LIN {X 0,Y 375.934,Z 136.466,A -85,B 0,C 180,E1 -12378.399,E2 -12378.399} C_VEL
LIN {X 0,Y 375.973,Z 136.465,A -85,B 0,C 180,E1 -12381.73,E2 -12381.73} C_VEL
LIN {X 0,Y 375.981,Z 136.466,A -85,B 0,C 180,E1 -12385.333,E2 -12385.333} C_VEL
LIN {X 0,Y 375.958,Z 136.463,A -85,B 0,C 180,E1 -12388.438,E2 -12388.438} C_VEL
LIN {X 0,Y 375.997,Z 136.458,A -85,B 0,C 180,E1 -12392.142,E2 -12392.142} C_VEL
LIN {X 0,Y 376.007,Z 136.459,A -85,B 0,C 180,E1 -12394.539,E2 -12394.539} C_VEL
LIN {X 0,Y 375.964,Z 136.462,A -85,B 0,C 180,E1 -12398.046,E2 -12398.046} C_VEL
LIN {X 0,Y 376.01,Z 136.457,A -85,B 0,C 180,E1 -12401.473,E2 -12401.473} C_VEL
LIN {X 0,Y 376.06,Z 136.455,A -85,B 0,C 180,E1 -12404.833,E2 -12404.833} C_VEL
LIN {X 0,Y 376.052,Z 136.454,A -85,B 0,C 180,E1 -12408.137,E2 -12408.137} C_VEL
LIN {X 0,Y 376.22,Z 136.432,A -85,B 0,C 180,E1 -12411.919,E2 -12411.919} C_VEL
LIN {X 0,Y 376.17,Z 136.439,A -85,B 0,C 180,E1 -12414.64,E2 -12414.64} C_VEL
LIN {X 0,Y 376.353,Z 136.417,A -85,B 0,C 180,E1 -12417.86,E2 -12417.86} C_VEL
LIN {X 0,Y 376.489,Z 136.403,A -85,B 0,C 180,E1 -12420,E2 -12420} C_VEL
LIN {X 0,Y 376.186,Z 136.435,A -85,B 0,C 180,E1 -12423.213,E2 -12423.213} C_VEL
LIN {X 0,Y 376.237,Z 136.429,A -85,B 0,C 180,E1 -12426.612,E2 -12426.612} C_VEL
LIN {X 0,Y 376.208,Z 136.432,A -85,B 0,C 180,E1 -12428.595,E2 -12428.595} C_VEL
LIN {X 0,Y 376.061,Z 136.454,A -85,B 0,C 180,E1 -12431.863,E2 -12431.863} C_VEL
LIN {X 0,Y 376.062,Z 136.453,A -85,B 0,C 180,E1 -12435.167,E2 -12435.167} C_VEL
LIN {X 0,Y 376.011,Z 136.457,A -85,B 0,C 180,E1 -12438.527,E2 -12438.527} C_VEL
LIN {X 0,Y 375.965,Z 136.463,A -85,B 0,C 180,E1 -12441.954,E2 -12441.954} C_VEL
LIN {X 0,Y 376.008,Z 136.46,A -85,B 0,C 180,E1 -12445.461,E2 -12445.461} C_VEL
LIN {X 0,Y 375.972,Z 136.467,A -85,B 0,C 180,E1 -12449.079,E2 -12449.079} C_VEL
LIN {X 0,Y 375.951,Z 136.471,A -85,B 0,C 180,E1 -12452.829,E2 -12452.829} C_VEL
LIN {X 0,Y 375.959,Z 136.464,A -85,B 0,C 180,E1 -12455.415,E2 -12455.415} C_VEL
LIN {X 0,Y 375.974,Z 136.464,A -85,B 0,C 180,E1 -12458.27,E2 -12458.27} C_VEL
LIN {X 0,Y 375.935,Z 136.466,A -85,B 0,C 180,E1 -12461.601,E2 -12461.601} C_VEL
LIN {X 0,Y 375.928,Z 136.467,A -85,B 0,C 180,E1 -12465.269,E2 -12465.269} C_VEL
LIN {X 0,Y 375.936,Z 136.471,A -85,B 0,C 180,E1 -12468.399,E2 -12468.399} C_VEL
LIN {X 0,Y 375.978,Z 136.463,A -85,B 0,C 180,E1 -12471.729,E2 -12471.729} C_VEL
LIN {X 0,Y 375.982,Z 136.461,A -85,B 0,C 180,E1 -12475.333,E2 -12475.333} C_VEL
LIN {X 0,Y 375.96,Z 136.464,A -85,B 0,C 180,E1 -12478.438,E2 -12478.438} C_VEL
LIN {X 0,Y 375.998,Z 136.46,A -85,B 0,C 180,E1 -12482.141,E2 -12482.141} C_VEL
LIN {X 0,Y 376.007,Z 136.457,A -85,B 0,C 180,E1 -12484.539,E2 -12484.539} C_VEL
LIN {X 0,Y 376.019,Z 136.597,A -85,B 0,C 180,E1 -12487.905,E2 -12487.905} C_VEL
LIN {X 0,Y 377.076,Z 142.753,A -85,B 0,C 180,E1 -12489.83,E2 -12489.83} C_VEL
LIN {X 0,Y 376.923,Z 150.73,A -85,B 0,C 180,E1 -12492.144,E2 -12492.144} C_VEL
LIN {X 0,Y 376.652,Z 155.114,A -85,B 0,C 180,E1 -12493.328,E2 -12493.328} C_VEL
LIN {X 0,Y 377.093,Z 157.794,A -85,B 0,C 180,E1 -12493.455,E2 -12493.455} C_VEL
LIN {X 0,Y 380.287,Z 175.775,A -85,B 0,C 180,E1 -12493.946,E2 -12493.946} C_VEL
LIN {X 0,Y 379.67,Z 231.165,A -85,B 0,C 180,E1 -12495.014,E2 -12495.014} C_VEL
LIN {X 0,Y 379.368,Z 241.032,A -85,B 0,C 180,E1 -12495.345,E2 -12495.345} C_VEL
LIN {X 0,Y 378.962,Z 252.164,A -85,B 0,C 180,E1 -12495.912,E2 -12495.912} C_VEL
LIN {X 0,Y 378.323,Z 263.011,A -85,B 0,C 180,E1 -12496.709,E2 -12496.709} C_VEL
LIN {X 0,Y 377.722,Z 271.413,A -85,B 0,C 180,E1 -12497.508,E2 -12497.508} C_VEL
LIN {X 0,Y 377.15,Z 279.343,A -85,B 0,C 180,E1 -12498.444,E2 -12498.444} C_VEL
LIN {X 0,Y 376.708,Z 285.037,A -85,B 0,C 180,E1 -12499.247,E2 -12499.247} C_VEL
LIN {X 0,Y 376.09,Z 291.396,A -85,B 0,C 180,E1 -12500.318,E2 -12500.318} C_VEL
LIN {X 0,Y 375.66,Z 296.679,A -85,B 0,C 180,E1 -12501.392,E2 -12501.392} C_VEL
LIN {X 0,Y 375.389,Z 301.089,A -85,B 0,C 180,E1 -12502.469,E2 -12502.469} C_VEL
LIN {X 0,Y 375.01,Z 306.274,A -85,B 0,C 180,E1 -12504.084,E2 -12504.084} C_VEL
LIN {X 0,Y 374.816,Z 308.937,A -85,B 0,C 180,E1 -12505.16,E2 -12505.16} C_VEL
LIN {X 0,Y 374.566,Z 311.853,A -85,B 0,C 180,E1 -12506.773,E2 -12506.773} C_VEL
LIN {X 0,Y 374.504,Z 313.128,A -85,B 0,C 180,E1 -12507.849,E2 -12507.849} C_VEL
LIN {X 0,Y 374.478,Z 313.933,A -85,B 0,C 180,E1 -12508.924,E2 -12508.924} C_VEL
LIN {X 0,Y 374.489,Z 314.239,A -85,B 0,C 180,E1 -12510,E2 -12510} C_VEL
LIN {X 0,Y 374.478,Z 313.964,A -85,B 0,C 180,E1 -12511.075,E2 -12511.075} C_VEL
LIN {X 0,Y 374.503,Z 313.22,A -85,B 0,C 180,E1 -12512.151,E2 -12512.151} C_VEL
LIN {X 0,Y 374.562,Z 312.007,A -85,B 0,C 180,E1 -12513.227,E2 -12513.227} C_VEL
LIN {X 0,Y 374.805,Z 309.155,A -85,B 0,C 180,E1 -12514.84,E2 -12514.84} C_VEL
LIN {X 0,Y 374.988,Z 306.561,A -85,B 0,C 180,E1 -12515.916,E2 -12515.916} C_VEL
LIN {X 0,Y 375.31,Z 302.523,A -85,B 0,C 180,E1 -12517.228,E2 -12517.228} C_VEL
LIN {X 0,Y 375.614,Z 297.127,A -85,B 0,C 180,E1 -12518.608,E2 -12518.608} C_VEL
LIN {X 0,Y 376.075,Z 291.933,A -85,B 0,C 180,E1 -12519.682,E2 -12519.682} C_VEL
LIN {X 0,Y 376.603,Z 285.676,A -85,B 0,C 180,E1 -12520.755,E2 -12520.755} C_VEL
LIN {X 0,Y 377.239,Z 278.068,A -85,B 0,C 180,E1 -12521.825,E2 -12521.825} C_VEL
LIN {X 0,Y 377.91,Z 268.598,A -85,B 0,C 180,E1 -12522.895,E2 -12522.895} C_VEL
LIN {X 0,Y 378.549,Z 259.324,A -85,B 0,C 180,E1 -12523.692,E2 -12523.692} C_VEL
LIN {X 0,Y 379.098,Z 250.369,A -85,B 0,C 180,E1 -12524.288,E2 -12524.288} C_VEL
LIN {X 0,Y 379.483,Z 241.034,A -85,B 0,C 180,E1 -12524.752,E2 -12524.752} C_VEL
LIN {X 0,Y 379.69,Z 233.061,A -85,B 0,C 180,E1 -12525.037,E2 -12525.037} C_VEL
LIN {X 0,Y 379.39,Z 227.278,A -85,B 0,C 180,E1 -12525.202,E2 -12525.202} C_VEL
LIN {X 0,Y 376.718,Z 217.95,A -85,B 0,C 180,E1 -12525.503,E2 -12525.503} C_VEL
LIN {X 0,Y 373.868,Z 208.608,A -85,B 0,C 180,E1 -12525.803,E2 -12525.803} C_VEL
LIN {X 0,Y 373.197,Z 202.789,A -85,B 0,C 180,E1 -12525.944,E2 -12525.944} C_VEL
LIN {X 0,Y 373.395,Z 176.209,A -85,B 0,C 180,E1 -12526.457,E2 -12526.457} C_VEL
LIN {X 0,Y 369.716,Z 155.569,A -85,B 0,C 180,E1 -12527.065,E2 -12527.065} C_VEL
LIN {X 0,Y 369.725,Z 154.415,A -85,B 0,C 180,E1 -12527.278,E2 -12527.278} C_VEL
LIN {X 0,Y 370.133,Z 145.161,A -85,B 0,C 180,E1 -12529.985,E2 -12529.985} C_VEL
LIN {X 0,Y 369.335,Z 139.36,A -85,B 0,C 180,E1 -12531.78,E2 -12531.78} C_VEL
LIN {X 0,Y 368.97,Z 137.432,A -85,B 0,C 180,E1 -12532.466,E2 -12532.466} C_VEL
LIN {X 0,Y 369,Z 137.332,A -85,B 0,C 180,E1 -12535.98,E2 -12535.98} C_VEL
LIN {X 0,Y 368.961,Z 137.336,A -85,B 0,C 180,E1 -12538.811,E2 -12538.811} C_VEL
LIN {X 0,Y 368.899,Z 137.348,A -85,B 0,C 180,E1 -12542.238,E2 -12542.238} C_VEL
LIN {X 0,Y 368.929,Z 137.339,A -85,B 0,C 180,E1 -12545.001,E2 -12545.001} C_VEL
LIN {X 0,Y 368.91,Z 137.342,A -85,B 0,C 180,E1 -12548.64,E2 -12548.64} C_VEL
LIN {X 0,Y 368.881,Z 137.349,A -85,B 0,C 180,E1 -12552.009,E2 -12552.009} C_VEL
LIN {X 0,Y 368.879,Z 137.346,A -85,B 0,C 180,E1 -12555.175,E2 -12555.175} C_VEL
LIN {X 0,Y 368.882,Z 137.346,A -85,B 0,C 180,E1 -12558.177,E2 -12558.177} C_VEL
LIN {X 0,Y 368.906,Z 137.347,A -85,B 0,C 180,E1 -12561.36,E2 -12561.36} C_VEL
LIN {X 0,Y 368.935,Z 137.342,A -85,B 0,C 180,E1 -12565.146,E2 -12565.146} C_VEL
LIN {X 0,Y 368.928,Z 137.344,A -85,B 0,C 180,E1 -12569.046,E2 -12569.046} C_VEL
LIN {X 0,Y 368.974,Z 137.335,A -85,B 0,C 180,E1 -12571.563,E2 -12571.563} C_VEL
LIN {X 0,Y 368.999,Z 137.33,A -85,B 0,C 180,E1 -12574.02,E2 -12574.02} C_VEL
LIN {X 0,Y 368.931,Z 137.339,A -85,B 0,C 180,E1 -12577.605,E2 -12577.605} C_VEL
LIN {X 0,Y 368.957,Z 137.338,A -85,B 0,C 180,E1 -12581.106,E2 -12581.106} C_VEL
LIN {X 0,Y 368.997,Z 137.336,A -85,B 0,C 180,E1 -12584.535,E2 -12584.535} C_VEL
LIN {X 0,Y 369.012,Z 137.33,A -85,B 0,C 180,E1 -12587.907,E2 -12587.907} C_VEL
LIN {X 0,Y 369.228,Z 137.303,A -85,B 0,C 180,E1 -12591.8,E2 -12591.8} C_VEL
LIN {X 0,Y 369.143,Z 137.315,A -85,B 0,C 180,E1 -12594.537,E2 -12594.537} C_VEL
LIN {X 0,Y 369.317,Z 137.294,A -85,B 0,C 180,E1 -12597.819,E2 -12597.819} C_VEL
LIN {X 0,Y 369.457,Z 137.279,A -85,B 0,C 180,E1 -12600,E2 -12600} C_VEL
LIN {X 0,Y 369.315,Z 137.294,A -85,B 0,C 180,E1 -12602.181,E2 -12602.181} C_VEL
LIN {X 0,Y 369.211,Z 137.304,A -85,B 0,C 180,E1 -12606.558,E2 -12606.558} C_VEL
LIN {X 0,Y 369.136,Z 137.313,A -85,B 0,C 180,E1 -12608.761,E2 -12608.761} C_VEL
LIN {X 0,Y 369.004,Z 137.331,A -85,B 0,C 180,E1 -12612.093,E2 -12612.093} C_VEL
LIN {X 0,Y 368.996,Z 137.336,A -85,B 0,C 180,E1 -12615.465,E2 -12615.465} C_VEL
LIN {X 0,Y 368.956,Z 137.338,A -85,B 0,C 180,E1 -12618.894,E2 -12618.894} C_VEL
LIN {X 0,Y 368.93,Z 137.339,A -85,B 0,C 180,E1 -12622.395,E2 -12622.395} C_VEL
LIN {X 0,Y 368.998,Z 137.33,A -85,B 0,C 180,E1 -12625.98,E2 -12625.98} C_VEL
LIN {X 0,Y 368.959,Z 137.341,A -85,B 0,C 180,E1 -12628.812,E2 -12628.812} C_VEL
LIN {X 0,Y 368.896,Z 137.344,A -85,B 0,C 180,E1 -12632.238,E2 -12632.238} C_VEL
LIN {X 0,Y 368.927,Z 137.342,A -85,B 0,C 180,E1 -12635.002,E2 -12635.002} C_VEL
LIN {X 0,Y 368.905,Z 137.346,A -85,B 0,C 180,E1 -12638.64,E2 -12638.64} C_VEL
LIN {X 0,Y 368.879,Z 137.348,A -85,B 0,C 180,E1 -12642.01,E2 -12642.01} C_VEL
LIN {X 0,Y 368.878,Z 137.345,A -85,B 0,C 180,E1 -12645.176,E2 -12645.176} C_VEL
LIN {X 0,Y 368.881,Z 137.351,A -85,B 0,C 180,E1 -12648.178,E2 -12648.178} C_VEL
LIN {X 0,Y 368.906,Z 137.342,A -85,B 0,C 180,E1 -12651.36,E2 -12651.36} C_VEL
LIN {X 0,Y 368.935,Z 137.338,A -85,B 0,C 180,E1 -12655.147,E2 -12655.147} C_VEL
LIN {X 0,Y 368.928,Z 137.34,A -85,B 0,C 180,E1 -12659.047,E2 -12659.047} C_VEL
LIN {X 0,Y 368.979,Z 137.338,A -85,B 0,C 180,E1 -12661.564,E2 -12661.564} C_VEL
LIN {X 0,Y 369.036,Z 137.429,A -85,B 0,C 180,E1 -12664.477,E2 -12664.477} C_VEL
LIN {X 0,Y 370.753,Z 147.316,A -85,B 0,C 180,E1 -12667.427,E2 -12667.427} C_VEL
LIN {X 0,Y 370.644,Z 152.562,A -85,B 0,C 180,E1 -12668.884,E2 -12668.884} C_VEL
LIN {X 0,Y 369.505,Z 167.651,A -85,B 0,C 180,E1 -12672.925,E2 -12672.925} C_VEL
LIN {X 0,Y 370.023,Z 171.195,A -85,B 0,C 180,E1 -12673.079,E2 -12673.079} C_VEL
LIN {X 0,Y 373.342,Z 194.927,A -85,B 0,C 180,E1 -12673.699,E2 -12673.699} C_VEL
LIN {X 0,Y 372.78,Z 244.263,A -85,B 0,C 180,E1 -12674.671,E2 -12674.671} C_VEL
LIN {X 0,Y 372.399,Z 253.93,A -85,B 0,C 180,E1 -12674.995,E2 -12674.995} C_VEL
LIN {X 0,Y 371.875,Z 263.95,A -85,B 0,C 180,E1 -12675.499,E2 -12675.499} C_VEL
LIN {X 0,Y 371.15,Z 275.333,A -85,B 0,C 180,E1 -12676.309,E2 -12676.309} C_VEL
LIN {X 0,Y 370.473,Z 283.91,A -85,B 0,C 180,E1 -12677.121,E2 -12677.121} C_VEL
LIN {X 0,Y 369.838,Z 291.982,A -85,B 0,C 180,E1 -12678.074,E2 -12678.074} C_VEL
LIN {X 0,Y 369.26,Z 298.649,A -85,B 0,C 180,E1 -12679.028,E2 -12679.028} C_VEL
LIN {X 0,Y 368.763,Z 304.98,A -85,B 0,C 180,E1 -12680.124,E2 -12680.124} C_VEL
LIN {X 0,Y 368.33,Z 310.239,A -85,B 0,C 180,E1 -12681.22,E2 -12681.22} C_VEL
LIN {X 0,Y 367.951,Z 314.625,A -85,B 0,C 180,E1 -12682.317,E2 -12682.317} C_VEL
LIN {X 0,Y 367.656,Z 319.143,A -85,B 0,C 180,E1 -12683.728,E2 -12683.728} C_VEL
LIN {X 0,Y 367.55,Z 322.442,A -85,B 0,C 180,E1 -12685.064,E2 -12685.064} C_VEL
LIN {X 0,Y 367.377,Z 325.342,A -85,B 0,C 180,E1 -12686.71,E2 -12686.71} C_VEL
LIN {X 0,Y 367.335,Z 326.592,A -85,B 0,C 180,E1 -12687.807,E2 -12687.807} C_VEL
LIN {X 0,Y 367.353,Z 327.369,A -85,B 0,C 180,E1 -12688.904,E2 -12688.904} C_VEL
LIN {X 0,Y 367.388,Z 327.664,A -85,B 0,C 180,E1 -12690,E2 -12690} C_VEL
LIN {X 0,Y 367.353,Z 327.365,A -85,B 0,C 180,E1 -12691.096,E2 -12691.096} C_VEL
LIN {X 0,Y 367.335,Z 326.58,A -85,B 0,C 180,E1 -12692.193,E2 -12692.193} C_VEL
LIN {X 0,Y 367.378,Z 325.322,A -85,B 0,C 180,E1 -12693.29,E2 -12693.29} C_VEL
LIN {X 0,Y 367.55,Z 322.414,A -85,B 0,C 180,E1 -12694.936,E2 -12694.936} C_VEL
LIN {X 0,Y 367.663,Z 319.081,A -85,B 0,C 180,E1 -12696.281,E2 -12696.281} C_VEL
LIN {X 0,Y 367.982,Z 313.614,A -85,B 0,C 180,E1 -12697.959,E2 -12697.959} C_VEL
LIN {X 0,Y 368.504,Z 307.744,A -85,B 0,C 180,E1 -12699.33,E2 -12699.33} C_VEL
LIN {X 0,Y 369.132,Z 300.275,A -85,B 0,C 180,E1 -12700.698,E2 -12700.698} C_VEL
LIN {X 0,Y 369.786,Z 292.911,A -85,B 0,C 180,E1 -12701.789,E2 -12701.789} C_VEL
LIN {X 0,Y 370.385,Z 285.023,A -85,B 0,C 180,E1 -12702.744,E2 -12702.744} C_VEL
LIN {X 0,Y 371.043,Z 276.687,A -85,B 0,C 180,E1 -12703.556,E2 -12703.556} C_VEL
LIN {X 0,Y 371.754,Z 266.036,A -85,B 0,C 180,E1 -12704.367,E2 -12704.367} C_VEL
LIN {X 0,Y 372.342,Z 254.431,A -85,B 0,C 180,E1 -12704.973,E2 -12704.973} C_VEL
LIN {X 0,Y 372.726,Z 244.695,A -85,B 0,C 180,E1 -12705.307,E2 -12705.307} C_VEL
LIN {X 0,Y 373.221,Z 192.86,A -85,B 0,C 180,E1 -12706.334,E2 -12706.334} C_VEL
LIN {X 0,Y 369.51,Z 167.924,A -85,B 0,C 180,E1 -12707.029,E2 -12707.029} C_VEL
LIN {X 0,Y 369.723,Z 163.572,A -85,B 0,C 180,E1 -12708.114,E2 -12708.114} C_VEL
LIN {X 0,Y 370.822,Z 150.112,A -85,B 0,C 180,E1 -12711.772,E2 -12711.772} C_VEL
LIN {X 0,Y 370.583,Z 146.203,A -85,B 0,C 180,E1 -12712.879,E2 -12712.879} C_VEL
LIN {X 0,Y 369.008,Z 137.41,A -85,B 0,C 180,E1 -12715.525,E2 -12715.525} C_VEL
LIN {X 0,Y 368.962,Z 137.337,A -85,B 0,C 180,E1 -12718.812,E2 -12718.812} C_VEL
LIN {X 0,Y 368.899,Z 137.349,A -85,B 0,C 180,E1 -12722.238,E2 -12722.238} C_VEL
LIN {X 0,Y 368.929,Z 137.339,A -85,B 0,C 180,E1 -12725.002,E2 -12725.002} C_VEL
LIN {X 0,Y 368.908,Z 137.342,A -85,B 0,C 180,E1 -12728.64,E2 -12728.64} C_VEL
LIN {X 0,Y 368.882,Z 137.349,A -85,B 0,C 180,E1 -12732.01,E2 -12732.01} C_VEL
LIN {X 0,Y 368.88,Z 137.346,A -85,B 0,C 180,E1 -12735.176,E2 -12735.176} C_VEL
LIN {X 0,Y 368.883,Z 137.346,A -85,B 0,C 180,E1 -12738.178,E2 -12738.178} C_VEL
LIN {X 0,Y 368.908,Z 137.346,A -85,B 0,C 180,E1 -12741.36,E2 -12741.36} C_VEL
LIN {X 0,Y 368.937,Z 137.341,A -85,B 0,C 180,E1 -12745.147,E2 -12745.147} C_VEL
LIN {X 0,Y 368.93,Z 137.343,A -85,B 0,C 180,E1 -12749.047,E2 -12749.047} C_VEL
LIN {X 0,Y 368.981,Z 137.334,A -85,B 0,C 180,E1 -12751.564,E2 -12751.564} C_VEL
LIN {X 0,Y 369.001,Z 137.33,A -85,B 0,C 180,E1 -12754.02,E2 -12754.02} C_VEL
LIN {X 0,Y 368.933,Z 137.339,A -85,B 0,C 180,E1 -12757.605,E2 -12757.605} C_VEL
LIN {X 0,Y 368.959,Z 137.338,A -85,B 0,C 180,E1 -12761.106,E2 -12761.106} C_VEL
LIN {X 0,Y 368.999,Z 137.335,A -85,B 0,C 180,E1 -12764.535,E2 -12764.535} C_VEL
LIN {X 0,Y 369.007,Z 137.33,A -85,B 0,C 180,E1 -12767.907,E2 -12767.907} C_VEL
LIN {X 0,Y 369.167,Z 137.311,A -85,B 0,C 180,E1 -12771.869,E2 -12771.869} C_VEL
LIN {X 0,Y 369.143,Z 137.316,A -85,B 0,C 180,E1 -12774.538,E2 -12774.538} C_VEL
LIN {X 0,Y 369.318,Z 137.293,A -85,B 0,C 180,E1 -12777.819,E2 -12777.819} C_VEL
LIN {X 0,Y 369.458,Z 137.278,A -85,B 0,C 180,E1 -12780,E2 -12780} C_VEL
LIN {X 0,Y 369.318,Z 137.295,A -85,B 0,C 180,E1 -12782.181,E2 -12782.181} C_VEL
LIN {X 0,Y 369.207,Z 137.304,A -85,B 0,C 180,E1 -12786.6,E2 -12786.6} C_VEL
LIN {X 0,Y 369.141,Z 137.312,A -85,B 0,C 180,E1 -12788.761,E2 -12788.761} C_VEL
LIN {X 0,Y 369.015,Z 137.33,A -85,B 0,C 180,E1 -12792.093,E2 -12792.093} C_VEL
LIN {X 0,Y 369.001,Z 137.336,A -85,B 0,C 180,E1 -12795.465,E2 -12795.465} C_VEL
LIN {X 0,Y 368.96,Z 137.337,A -85,B 0,C 180,E1 -12798.894,E2 -12798.894} C_VEL
LIN {X 0,Y 368.934,Z 137.338,A -85,B 0,C 180,E1 -12802.395,E2 -12802.395} C_VEL
LIN {X 0,Y 369.002,Z 137.33,A -85,B 0,C 180,E1 -12805.98,E2 -12805.98} C_VEL
LIN {X 0,Y 368.961,Z 137.339,A -85,B 0,C 180,E1 -12808.811,E2 -12808.811} C_VEL
LIN {X 0,Y 368.9,Z 137.343,A -85,B 0,C 180,E1 -12812.238,E2 -12812.238} C_VEL
LIN {X 0,Y 368.931,Z 137.342,A -85,B 0,C 180,E1 -12815.001,E2 -12815.001} C_VEL
LIN {X 0,Y 368.909,Z 137.347,A -85,B 0,C 180,E1 -12818.64,E2 -12818.64} C_VEL
LIN {X 0,Y 368.883,Z 137.346,A -85,B 0,C 180,E1 -12822.009,E2 -12822.009} C_VEL
LIN {X 0,Y 368.881,Z 137.345,A -85,B 0,C 180,E1 -12825.176,E2 -12825.176} C_VEL
LIN {X 0,Y 368.885,Z 137.35,A -85,B 0,C 180,E1 -12828.178,E2 -12828.178} C_VEL
LIN {X 0,Y 368.912,Z 137.341,A -85,B 0,C 180,E1 -12831.359,E2 -12831.359} C_VEL
LIN {X 0,Y 368.939,Z 137.338,A -85,B 0,C 180,E1 -12835.147,E2 -12835.147} C_VEL
LIN {X 0,Y 368.931,Z 137.339,A -85,B 0,C 180,E1 -12839.046,E2 -12839.046} C_VEL
LIN {X 0,Y 368.982,Z 137.336,A -85,B 0,C 180,E1 -12841.564,E2 -12841.564} C_VEL
LIN {X 0,Y 369.002,Z 137.332,A -85,B 0,C 180,E1 -12844.02,E2 -12844.02} C_VEL
LIN {X 0,Y 368.992,Z 137.519,A -85,B 0,C 180,E1 -12847.719,E2 -12847.719} C_VEL
LIN {X 0,Y 369.966,Z 142.869,A -85,B 0,C 180,E1 -12849.425,E2 -12849.425} C_VEL
LIN {X 0,Y 370.054,Z 148.689,A -85,B 0,C 180,E1 -12851.164,E2 -12851.164} C_VEL
LIN {X 0,Y 369.693,Z 155.057,A -85,B 0,C 180,E1 -12852.98,E2 -12852.98} C_VEL
LIN {X 0,Y 369.947,Z 156.928,A -85,B 0,C 180,E1 -12853.106,E2 -12853.106} C_VEL
LIN {X 0,Y 373.491,Z 177.315,A -85,B 0,C 180,E1 -12853.673,E2 -12853.673} C_VEL
LIN {X 0,Y 372.834,Z 231.311,A -85,B 0,C 180,E1 -12854.733,E2 -12854.733} C_VEL
LIN {X 0,Y 372.518,Z 241.172,A -85,B 0,C 180,E1 -12855.07,E2 -12855.07} C_VEL
LIN {X 0,Y 372.154,Z 251.108,A -85,B 0,C 180,E1 -12855.579,E2 -12855.579} C_VEL
LIN {X 0,Y 371.532,Z 261.637,A -85,B 0,C 180,E1 -12856.322,E2 -12856.322} C_VEL
LIN {X 0,Y 370.785,Z 271.546,A -85,B 0,C 180,E1 -12857.27,E2 -12857.27} C_VEL
LIN {X 0,Y 370.197,Z 279.475,A -85,B 0,C 180,E1 -12858.224,E2 -12858.224} C_VEL
LIN {X 0,Y 369.728,Z 285.169,A -85,B 0,C 180,E1 -12859.042,E2 -12859.042} C_VEL
LIN {X 0,Y 369.104,Z 291.526,A -85,B 0,C 180,E1 -12860.132,E2 -12860.132} C_VEL
LIN {X 0,Y 368.549,Z 297.979,A -85,B 0,C 180,E1 -12861.501,E2 -12861.501} C_VEL
LIN {X 0,Y 368.213,Z 303.127,A -85,B 0,C 180,E1 -12862.874,E2 -12862.874} C_VEL
LIN {X 0,Y 367.848,Z 307.89,A -85,B 0,C 180,E1 -12864.518,E2 -12864.518} C_VEL
LIN {X 0,Y 367.647,Z 310.213,A -85,B 0,C 180,E1 -12865.614,E2 -12865.614} C_VEL
LIN {X 0,Y 367.483,Z 311.982,A -85,B 0,C 180,E1 -12866.711,E2 -12866.711} C_VEL
LIN {X 0,Y 367.407,Z 313.257,A -85,B 0,C 180,E1 -12867.807,E2 -12867.807} C_VEL
LIN {X 0,Y 367.379,Z 314.062,A -85,B 0,C 180,E1 -12868.904,E2 -12868.904} C_VEL
LIN {X 0,Y 367.391,Z 314.368,A -85,B 0,C 180,E1 -12870,E2 -12870} C_VEL
LIN {X 0,Y 367.379,Z 314.092,A -85,B 0,C 180,E1 -12871.096,E2 -12871.096} C_VEL
LIN {X 0,Y 367.406,Z 313.348,A -85,B 0,C 180,E1 -12872.192,E2 -12872.192} C_VEL
LIN {X 0,Y 367.479,Z 312.135,A -85,B 0,C 180,E1 -12873.289,E2 -12873.289} C_VEL
LIN {X 0,Y 367.748,Z 309.283,A -85,B 0,C 180,E1 -12874.933,E2 -12874.933} C_VEL
LIN {X 0,Y 367.931,Z 306.688,A -85,B 0,C 180,E1 -12876.03,E2 -12876.03} C_VEL
LIN {X 0,Y 368.249,Z 302.862,A -85,B 0,C 180,E1 -12877.306,E2 -12877.306} C_VEL
LIN {X 0,Y 368.518,Z 298.423,A -85,B 0,C 180,E1 -12878.499,E2 -12878.499} C_VEL
LIN {X 0,Y 368.952,Z 293.475,A -85,B 0,C 180,E1 -12879.594,E2 -12879.594} C_VEL
LIN {X 0,Y 369.499,Z 287.501,A -85,B 0,C 180,E1 -12880.687,E2 -12880.687} C_VEL
LIN {X 0,Y 370.137,Z 280.23,A -85,B 0,C 180,E1 -12881.777,E2 -12881.777} C_VEL
LIN {X 0,Y 370.699,Z 273.686,A -85,B 0,C 180,E1 -12882.593,E2 -12882.593} C_VEL
LIN {X 0,Y 371.188,Z 267.259,A -85,B 0,C 180,E1 -12883.272,E2 -12883.272} C_VEL
LIN {X 0,Y 371.651,Z 259.446,A -85,B 0,C 180,E1 -12883.951,E2 -12883.951} C_VEL
LIN {X 0,Y 372.235,Z 250.488,A -85,B 0,C 180,E1 -12884.557,E2 -12884.557} C_VEL
LIN {X 0,Y 372.627,Z 241.15,A -85,B 0,C 180,E1 -12885.03,E2 -12885.03} C_VEL
LIN {X 0,Y 372.896,Z 231.672,A -85,B 0,C 180,E1 -12885.358,E2 -12885.358} C_VEL
LIN {X 0,Y 373.197,Z 202.789,A -85,B 0,C 180,E1 -12885.944,E2 -12885.944} C_VEL
LIN {X 0,Y 372.692,Z 196.967,A -85,B 0,C 180,E1 -12886.081,E2 -12886.081} C_VEL
LIN {X 0,Y 370.309,Z 187.56,A -85,B 0,C 180,E1 -12886.374,E2 -12886.374} C_VEL
LIN {X 0,Y 367.889,Z 180.12,A -85,B 0,C 180,E1 -12886.634,E2 -12886.634} C_VEL
LIN {X 0,Y 365.864,Z 172.558,A -85,B 0,C 180,E1 -12886.881,E2 -12886.881} C_VEL
LIN {X 0,Y 362.811,Z 155.749,A -85,B 0,C 180,E1 -12887.394,E2 -12887.394} C_VEL
LIN {X 0,Y 362.784,Z 154.536,A -85,B 0,C 180,E1 -12887.619,E2 -12887.619} C_VEL
LIN {X 0,Y 363.162,Z 147.216,A -85,B 0,C 180,E1 -12889.795,E2 -12889.795} C_VEL
LIN {X 0,Y 362.52,Z 141.401,A -85,B 0,C 180,E1 -12891.613,E2 -12891.613} C_VEL
LIN {X 0,Y 361.936,Z 138.321,A -85,B 0,C 180,E1 -12892.663,E2 -12892.663} C_VEL
LIN {X 0,Y 361.943,Z 138.212,A -85,B 0,C 180,E1 -12896.721,E2 -12896.721} C_VEL
LIN {X 0,Y 361.875,Z 138.223,A -85,B 0,C 180,E1 -12900.328,E2 -12900.328} C_VEL
LIN {X 0,Y 361.855,Z 138.224,A -85,B 0,C 180,E1 -12904.28,E2 -12904.28} C_VEL
LIN {X 0,Y 361.865,Z 138.219,A -85,B 0,C 180,E1 -12907.223,E2 -12907.223} C_VEL
LIN {X 0,Y 361.835,Z 138.222,A -85,B 0,C 180,E1 -12910.755,E2 -12910.755} C_VEL
LIN {X 0,Y 361.816,Z 138.226,A -85,B 0,C 180,E1 -12914.368,E2 -12914.368} C_VEL
LIN {X 0,Y 361.835,Z 138.228,A -85,B 0,C 180,E1 -12917.568,E2 -12917.568} C_VEL
LIN {X 0,Y 361.867,Z 138.22,A -85,B 0,C 180,E1 -12920.973,E2 -12920.973} C_VEL
LIN {X 0,Y 361.873,Z 138.218,A -85,B 0,C 180,E1 -12924.655,E2 -12924.655} C_VEL
LIN {X 0,Y 361.836,Z 138.223,A -85,B 0,C 180,E1 -12928.37,E2 -12928.37} C_VEL
LIN {X 0,Y 361.899,Z 138.219,A -85,B 0,C 180,E1 -12930.955,E2 -12930.955} C_VEL
LIN {X 0,Y 361.953,Z 138.21,A -85,B 0,C 180,E1 -12933.475,E2 -12933.475} C_VEL
LIN {X 0,Y 361.889,Z 138.219,A -85,B 0,C 180,E1 -12937.144,E2 -12937.144} C_VEL
LIN {X 0,Y 361.905,Z 138.22,A -85,B 0,C 180,E1 -12940.723,E2 -12940.723} C_VEL
LIN {X 0,Y 361.931,Z 138.212,A -85,B 0,C 180,E1 -12943.066,E2 -12943.066} C_VEL
LIN {X 0,Y 361.999,Z 138.208,A -85,B 0,C 180,E1 -12946.528,E2 -12946.528} C_VEL
LIN {X 0,Y 362.035,Z 138.2,A -85,B 0,C 180,E1 -12949.938,E2 -12949.938} C_VEL
LIN {X 0,Y 362.15,Z 138.189,A -85,B 0,C 180,E1 -12952.192,E2 -12952.192} C_VEL
LIN {X 0,Y 362.117,Z 138.191,A -85,B 0,C 180,E1 -12954.431,E2 -12954.431} C_VEL
LIN {X 0,Y 362.281,Z 138.17,A -85,B 0,C 180,E1 -12957.776,E2 -12957.776} C_VEL
LIN {X 0,Y 362.426,Z 138.155,A -85,B 0,C 180,E1 -12960,E2 -12960} C_VEL
LIN {X 0,Y 362.279,Z 138.17,A -85,B 0,C 180,E1 -12962.223,E2 -12962.223} C_VEL
LIN {X 0,Y 362.174,Z 138.18,A -85,B 0,C 180,E1 -12966.686,E2 -12966.686} C_VEL
LIN {X 0,Y 362.072,Z 138.193,A -85,B 0,C 180,E1 -12968.933,E2 -12968.933} C_VEL
LIN {X 0,Y 361.958,Z 138.207,A -85,B 0,C 180,E1 -12972.332,E2 -12972.332} C_VEL
LIN {X 0,Y 361.96,Z 138.207,A -85,B 0,C 180,E1 -12974.62,E2 -12974.62} C_VEL
LIN {X 0,Y 361.954,Z 138.208,A -85,B 0,C 180,E1 -12978.099,E2 -12978.099} C_VEL
LIN {X 0,Y 361.89,Z 138.217,A -85,B 0,C 180,E1 -12981.653,E2 -12981.653} C_VEL
LIN {X 0,Y 361.926,Z 138.214,A -85,B 0,C 180,E1 -12985.29,E2 -12985.29} C_VEL
LIN {X 0,Y 361.916,Z 138.212,A -85,B 0,C 180,E1 -12987.778,E2 -12987.778} C_VEL
LIN {X 0,Y 361.844,Z 138.223,A -85,B 0,C 180,E1 -12991.285,E2 -12991.285} C_VEL
LIN {X 0,Y 361.852,Z 138.223,A -85,B 0,C 180,E1 -12994.28,E2 -12994.28} C_VEL
LIN {X 0,Y 361.861,Z 138.22,A -85,B 0,C 180,E1 -12997.223,E2 -12997.223} C_VEL
LIN {X 0,Y 361.833,Z 138.225,A -85,B 0,C 180,E1 -13000.755,E2 -13000.755} C_VEL
LIN {X 0,Y 361.816,Z 138.23,A -85,B 0,C 180,E1 -13004.369,E2 -13004.369} C_VEL
LIN {X 0,Y 361.834,Z 138.224,A -85,B 0,C 180,E1 -13007.568,E2 -13007.568} C_VEL
LIN {X 0,Y 361.867,Z 138.218,A -85,B 0,C 180,E1 -13010.974,E2 -13010.974} C_VEL
LIN {X 0,Y 361.873,Z 138.218,A -85,B 0,C 180,E1 -13014.655,E2 -13014.655} C_VEL
LIN {X 0,Y 361.836,Z 138.223,A -85,B 0,C 180,E1 -13018.371,E2 -13018.371} C_VEL
LIN {X 0,Y 361.899,Z 138.215,A -85,B 0,C 180,E1 -13020.956,E2 -13020.956} C_VEL
LIN {X 0,Y 361.981,Z 138.414,A -85,B 0,C 180,E1 -13024.291,E2 -13024.291} C_VEL
LIN {X 0,Y 363.723,Z 148.237,A -85,B 0,C 180,E1 -13027.267,E2 -13027.267} C_VEL
LIN {X 0,Y 363.899,Z 150.685,A -85,B 0,C 180,E1 -13027.975,E2 -13027.975} C_VEL
LIN {X 0,Y 362.736,Z 164.089,A -85,B 0,C 180,E1 -13031.69,E2 -13031.69} C_VEL
LIN {X 0,Y 362.538,Z 167.524,A -85,B 0,C 180,E1 -13032.587,E2 -13032.587} C_VEL
LIN {X 0,Y 363.088,Z 171.264,A -85,B 0,C 180,E1 -13032.749,E2 -13032.749} C_VEL
LIN {X 0,Y 366.537,Z 195.003,A -85,B 0,C 180,E1 -13033.391,E2 -13033.391} C_VEL
LIN {X 0,Y 365.95,Z 244.201,A -85,B 0,C 180,E1 -13034.379,E2 -13034.379} C_VEL
LIN {X 0,Y 365.553,Z 253.811,A -85,B 0,C 180,E1 -13034.708,E2 -13034.708} C_VEL
LIN {X 0,Y 365.024,Z 263.829,A -85,B 0,C 180,E1 -13035.22,E2 -13035.22} C_VEL
LIN {X 0,Y 364.249,Z 275.209,A -85,B 0,C 180,E1 -13036.044,E2 -13036.044} C_VEL
LIN {X 0,Y 363.567,Z 283.786,A -85,B 0,C 180,E1 -13036.872,E2 -13036.872} C_VEL
LIN {X 0,Y 362.885,Z 291.856,A -85,B 0,C 180,E1 -13037.842,E2 -13037.842} C_VEL
LIN {X 0,Y 362.298,Z 298.523,A -85,B 0,C 180,E1 -13038.815,E2 -13038.815} C_VEL
LIN {X 0,Y 361.731,Z 304.852,A -85,B 0,C 180,E1 -13039.93,E2 -13039.93} C_VEL
LIN {X 0,Y 361.288,Z 310.112,A -85,B 0,C 180,E1 -13041.047,E2 -13041.047} C_VEL
LIN {X 0,Y 360.92,Z 314.498,A -85,B 0,C 180,E1 -13042.166,E2 -13042.166} C_VEL
LIN {X 0,Y 360.556,Z 319.467,A -85,B 0,C 180,E1 -13043.771,E2 -13043.771} C_VEL
LIN {X 0,Y 360.45,Z 322.314,A -85,B 0,C 180,E1 -13044.967,E2 -13044.967} C_VEL
LIN {X 0,Y 360.301,Z 325.214,A -85,B 0,C 180,E1 -13046.646,E2 -13046.646} C_VEL
LIN {X 0,Y 360.241,Z 326.463,A -85,B 0,C 180,E1 -13047.764,E2 -13047.764} C_VEL
LIN {X 0,Y 360.253,Z 327.241,A -85,B 0,C 180,E1 -13048.882,E2 -13048.882} C_VEL
LIN {X 0,Y 360.289,Z 327.535,A -85,B 0,C 180,E1 -13050,E2 -13050} C_VEL
LIN {X 0,Y 360.253,Z 327.237,A -85,B 0,C 180,E1 -13051.118,E2 -13051.118} C_VEL
LIN {X 0,Y 360.241,Z 326.451,A -85,B 0,C 180,E1 -13052.236,E2 -13052.236} C_VEL
LIN {X 0,Y 360.301,Z 325.193,A -85,B 0,C 180,E1 -13053.355,E2 -13053.355} C_VEL
LIN {X 0,Y 360.45,Z 322.284,A -85,B 0,C 180,E1 -13055.034,E2 -13055.034} C_VEL
LIN {X 0,Y 360.556,Z 319.43,A -85,B 0,C 180,E1 -13056.229,E2 -13056.229} C_VEL
LIN {X 0,Y 360.866,Z 314.445,A -85,B 0,C 180,E1 -13057.836,E2 -13057.836} C_VEL
LIN {X 0,Y 361.476,Z 307.613,A -85,B 0,C 180,E1 -13059.513,E2 -13059.513} C_VEL
LIN {X 0,Y 362.137,Z 300.144,A -85,B 0,C 180,E1 -13060.907,E2 -13060.907} C_VEL
LIN {X 0,Y 362.808,Z 292.779,A -85,B 0,C 180,E1 -13062.019,E2 -13062.019} C_VEL
LIN {X 0,Y 363.464,Z 284.891,A -85,B 0,C 180,E1 -13062.99,E2 -13062.99} C_VEL
LIN {X 0,Y 364.144,Z 276.555,A -85,B 0,C 180,E1 -13063.818,E2 -13063.818} C_VEL
LIN {X 0,Y 364.888,Z 265.902,A -85,B 0,C 180,E1 -13064.643,E2 -13064.643} C_VEL
LIN {X 0,Y 365.471,Z 254.292,A -85,B 0,C 180,E1 -13065.261,E2 -13065.261} C_VEL
LIN {X 0,Y 365.899,Z 244.552,A -85,B 0,C 180,E1 -13065.599,E2 -13065.599} C_VEL
LIN {X 0,Y 366.33,Z 192.983,A -85,B 0,C 180,E1 -13066.644,E2 -13066.644} C_VEL
LIN {X 0,Y 362.563,Z 167.79,A -85,B 0,C 180,E1 -13067.365,E2 -13067.365} C_VEL
LIN {X 0,Y 362.818,Z 162.712,A -85,B 0,C 180,E1 -13068.676,E2 -13068.676} C_VEL
LIN {X 0,Y 363.853,Z 150.699,A -85,B 0,C 180,E1 -13072.007,E2 -13072.007} C_VEL
LIN {X 0,Y 363.195,Z 145.014,A -85,B 0,C 180,E1 -13073.674,E2 -13073.674} C_VEL
LIN {X 0,Y 361.988,Z 138.248,A -85,B 0,C 180,E1 -13075.787,E2 -13075.787} C_VEL
LIN {X 0,Y 361.913,Z 138.213,A -85,B 0,C 180,E1 -13079.09,E2 -13079.09} C_VEL
LIN {X 0,Y 361.849,Z 138.221,A -85,B 0,C 180,E1 -13082.945,E2 -13082.945} C_VEL
LIN {X 0,Y 361.868,Z 138.22,A -85,B 0,C 180,E1 -13085.637,E2 -13085.637} C_VEL
LIN {X 0,Y 361.869,Z 138.218,A -85,B 0,C 180,E1 -13089.027,E2 -13089.027} C_VEL
LIN {X 0,Y 361.837,Z 138.222,A -85,B 0,C 180,E1 -13092.829,E2 -13092.829} C_VEL
LIN {X 0,Y 361.819,Z 138.228,A -85,B 0,C 180,E1 -13095.947,E2 -13095.947} C_VEL
LIN {X 0,Y 361.836,Z 138.225,A -85,B 0,C 180,E1 -13099.245,E2 -13099.245} C_VEL
LIN {X 0,Y 361.864,Z 138.219,A -85,B 0,C 180,E1 -13102.777,E2 -13102.777} C_VEL
LIN {X 0,Y 361.855,Z 138.223,A -85,B 0,C 180,E1 -13105.72,E2 -13105.72} C_VEL
LIN {X 0,Y 361.875,Z 138.219,A -85,B 0,C 180,E1 -13109.672,E2 -13109.672} C_VEL
LIN {X 0,Y 361.956,Z 138.21,A -85,B 0,C 180,E1 -13113.475,E2 -13113.475} C_VEL
LIN {X 0,Y 361.891,Z 138.219,A -85,B 0,C 180,E1 -13117.145,E2 -13117.145} C_VEL
LIN {X 0,Y 361.908,Z 138.219,A -85,B 0,C 180,E1 -13120.724,E2 -13120.724} C_VEL
LIN {X 0,Y 361.934,Z 138.213,A -85,B 0,C 180,E1 -13123.066,E2 -13123.066} C_VEL
LIN {X 0,Y 362.001,Z 138.208,A -85,B 0,C 180,E1 -13126.528,E2 -13126.528} C_VEL
LIN {X 0,Y 362.033,Z 138.199,A -85,B 0,C 180,E1 -13129.938,E2 -13129.938} C_VEL
LIN {X 0,Y 362.163,Z 138.182,A -85,B 0,C 180,E1 -13133.314,E2 -13133.314} C_VEL
LIN {X 0,Y 362.282,Z 138.169,A -85,B 0,C 180,E1 -13137.777,E2 -13137.777} C_VEL
LIN {X 0,Y 362.428,Z 138.154,A -85,B 0,C 180,E1 -13140,E2 -13140} C_VEL
LIN {X 0,Y 362.282,Z 138.171,A -85,B 0,C 180,E1 -13142.224,E2 -13142.224} C_VEL
LIN {X 0,Y 362.174,Z 138.18,A -85,B 0,C 180,E1 -13146.686,E2 -13146.686} C_VEL
LIN {X 0,Y 362.077,Z 138.192,A -85,B 0,C 180,E1 -13148.933,E2 -13148.933} C_VEL
LIN {X 0,Y 361.968,Z 138.206,A -85,B 0,C 180,E1 -13152.332,E2 -13152.332} C_VEL
LIN {X 0,Y 361.964,Z 138.206,A -85,B 0,C 180,E1 -13154.62,E2 -13154.62} C_VEL
LIN {X 0,Y 361.958,Z 138.208,A -85,B 0,C 180,E1 -13158.1,E2 -13158.1} C_VEL
LIN {X 0,Y 361.894,Z 138.217,A -85,B 0,C 180,E1 -13161.653,E2 -13161.653} C_VEL
LIN {X 0,Y 361.93,Z 138.215,A -85,B 0,C 180,E1 -13165.29,E2 -13165.29} C_VEL
LIN {X 0,Y 361.916,Z 138.213,A -85,B 0,C 180,E1 -13167.779,E2 -13167.779} C_VEL
LIN {X 0,Y 361.848,Z 138.223,A -85,B 0,C 180,E1 -13171.285,E2 -13171.285} C_VEL
LIN {X 0,Y 361.856,Z 138.221,A -85,B 0,C 180,E1 -13174.28,E2 -13174.28} C_VEL
LIN {X 0,Y 361.865,Z 138.22,A -85,B 0,C 180,E1 -13177.223,E2 -13177.223} C_VEL
LIN {X 0,Y 361.837,Z 138.226,A -85,B 0,C 180,E1 -13180.755,E2 -13180.755} C_VEL
LIN {X 0,Y 361.819,Z 138.23,A -85,B 0,C 180,E1 -13184.368,E2 -13184.368} C_VEL
LIN {X 0,Y 361.838,Z 138.223,A -85,B 0,C 180,E1 -13187.568,E2 -13187.568} C_VEL
LIN {X 0,Y 361.873,Z 138.218,A -85,B 0,C 180,E1 -13190.973,E2 -13190.973} C_VEL
LIN {X 0,Y 361.876,Z 138.218,A -85,B 0,C 180,E1 -13194.655,E2 -13194.655} C_VEL
LIN {X 0,Y 361.84,Z 138.223,A -85,B 0,C 180,E1 -13198.371,E2 -13198.371} C_VEL
LIN {X 0,Y 361.902,Z 138.214,A -85,B 0,C 180,E1 -13200.955,E2 -13200.955} C_VEL
LIN {X 0,Y 361.956,Z 138.211,A -85,B 0,C 180,E1 -13203.475,E2 -13203.475} C_VEL
LIN {X 0,Y 361.925,Z 138.36,A -85,B 0,C 180,E1 -13207.486,E2 -13207.486} C_VEL
LIN {X 0,Y 363.053,Z 144.921,A -85,B 0,C 180,E1 -13209.608,E2 -13209.608} C_VEL
LIN {X 0,Y 363.017,Z 151.38,A -85,B 0,C 180,E1 -13211.557,E2 -13211.557} C_VEL
LIN {X 0,Y 362.764,Z 155.186,A -85,B 0,C 180,E1 -13212.645,E2 -13212.645} C_VEL
LIN {X 0,Y 363.014,Z 157.066,A -85,B 0,C 180,E1 -13212.773,E2 -13212.773} C_VEL
LIN {X 0,Y 366.689,Z 177.78,A -85,B 0,C 180,E1 -13213.368,E2 -13213.368} C_VEL
LIN {X 0,Y 366.003,Z 231.458,A -85,B 0,C 180,E1 -13214.441,E2 -13214.441} C_VEL
LIN {X 0,Y 365.688,Z 241.311,A -85,B 0,C 180,E1 -13214.784,E2 -13214.784} C_VEL
LIN {X 0,Y 365.297,Z 251.244,A -85,B 0,C 180,E1 -13215.302,E2 -13215.302} C_VEL
LIN {X 0,Y 364.652,Z 261.771,A -85,B 0,C 180,E1 -13216.059,E2 -13216.059} C_VEL
LIN {X 0,Y 363.863,Z 271.679,A -85,B 0,C 180,E1 -13217.024,E2 -13217.024} C_VEL
LIN {X 0,Y 363.246,Z 279.607,A -85,B 0,C 180,E1 -13217.995,E2 -13217.995} C_VEL
LIN {X 0,Y 362.75,Z 285.3,A -85,B 0,C 180,E1 -13218.828,E2 -13218.828} C_VEL
LIN {X 0,Y 362.131,Z 291.657,A -85,B 0,C 180,E1 -13219.941,E2 -13219.941} C_VEL
LIN {X 0,Y 361.615,Z 296.94,A -85,B 0,C 180,E1 -13221.055,E2 -13221.055} C_VEL
LIN {X 0,Y 361.309,Z 301.349,A -85,B 0,C 180,E1 -13222.174,E2 -13222.174} C_VEL
LIN {X 0,Y 360.933,Z 305.781,A -85,B 0,C 180,E1 -13223.573,E2 -13223.573} C_VEL
LIN {X 0,Y 360.705,Z 309.195,A -85,B 0,C 180,E1 -13224.97,E2 -13224.97} C_VEL
LIN {X 0,Y 360.403,Z 312.111,A -85,B 0,C 180,E1 -13226.646,E2 -13226.646} C_VEL
LIN {X 0,Y 360.312,Z 313.386,A -85,B 0,C 180,E1 -13227.764,E2 -13227.764} C_VEL
LIN {X 0,Y 360.281,Z 314.19,A -85,B 0,C 180,E1 -13228.882,E2 -13228.882} C_VEL
LIN {X 0,Y 360.292,Z 314.496,A -85,B 0,C 180,E1 -13230,E2 -13230} C_VEL
LIN {X 0,Y 360.281,Z 314.22,A -85,B 0,C 180,E1 -13231.117,E2 -13231.117} C_VEL
LIN {X 0,Y 360.311,Z 313.476,A -85,B 0,C 180,E1 -13232.235,E2 -13232.235} C_VEL
LIN {X 0,Y 360.399,Z 312.263,A -85,B 0,C 180,E1 -13233.354,E2 -13233.354} C_VEL
LIN {X 0,Y 360.691,Z 309.41,A -85,B 0,C 180,E1 -13235.03,E2 -13235.03} C_VEL
LIN {X 0,Y 360.881,Z 306.266,A -85,B 0,C 180,E1 -13236.353,E2 -13236.353} C_VEL
LIN {X 0,Y 361.266,Z 301.707,A -85,B 0,C 180,E1 -13237.826,E2 -13237.826} C_VEL
LIN {X 0,Y 361.69,Z 296.211,A -85,B 0,C 180,E1 -13239.224,E2 -13239.224} C_VEL
LIN {X 0,Y 362.395,Z 289.305,A -85,B 0,C 180,E1 -13240.616,E2 -13240.616} C_VEL
LIN {X 0,Y 363.11,Z 281.374,A -85,B 0,C 180,E1 -13241.867,E2 -13241.867} C_VEL
LIN {X 0,Y 363.788,Z 273.81,A -85,B 0,C 180,E1 -13242.836,E2 -13242.836} C_VEL
LIN {X 0,Y 364.301,Z 267.381,A -85,B 0,C 180,E1 -13243.527,E2 -13243.527} C_VEL
LIN {X 0,Y 364.778,Z 259.568,A -85,B 0,C 180,E1 -13244.22,E2 -13244.22} C_VEL
LIN {X 0,Y 365.381,Z 250.608,A -85,B 0,C 180,E1 -13244.836,E2 -13244.836} C_VEL
LIN {X 0,Y 365.788,Z 241.267,A -85,B 0,C 180,E1 -13245.318,E2 -13245.318} C_VEL
LIN {X 0,Y 366.068,Z 231.87,A -85,B 0,C 180,E1 -13245.65,E2 -13245.65} C_VEL
LIN {X 0,Y 366.628,Z 185.349,A -85,B 0,C 180,E1 -13246.589,E2 -13246.589} C_VEL
LIN {X 0,Y 366.53,Z 176.327,A -85,B 0,C 180,E1 -13246.774,E2 -13246.774} C_VEL
LIN {X 0,Y 365.864,Z 172.558,A -85,B 0,C 180,E1 -13246.881,E2 -13246.881} C_VEL
LIN {X 0,Y 364.2,Z 167.235,A -85,B 0,C 180,E1 -13247.104,E2 -13247.104} C_VEL
LIN {X 0,Y 361.032,Z 160.87,A -85,B 0,C 180,E1 -13247.575,E2 -13247.575} C_VEL
LIN {X 0,Y 357.959,Z 155.367,A -85,B 0,C 180,E1 -13248.25,E2 -13248.25} C_VEL
LIN {X 0,Y 356.428,Z 151.842,A -85,B 0,C 180,E1 -13248.908,E2 -13248.908} C_VEL
LIN {X 0,Y 356.123,Z 149.889,A -85,B 0,C 180,E1 -13249.416,E2 -13249.416} C_VEL
LIN {X 0,Y 355.788,Z 144,A -85,B 0,C 180,E1 -13251.261,E2 -13251.261} C_VEL
LIN {X 0,Y 354.885,Z 139.209,A -85,B 0,C 180,E1 -13252.87,E2 -13252.87} C_VEL
LIN {X 0,Y 354.899,Z 139.088,A -85,B 0,C 180,E1 -13255.827,E2 -13255.827} C_VEL
LIN {X 0,Y 354.854,Z 139.093,A -85,B 0,C 180,E1 -13259.678,E2 -13259.678} C_VEL
LIN {X 0,Y 354.806,Z 139.1,A -85,B 0,C 180,E1 -13263.702,E2 -13263.702} C_VEL
LIN {X 0,Y 354.799,Z 139.101,A -85,B 0,C 180,E1 -13266.459,E2 -13266.459} C_VEL
LIN {X 0,Y 354.824,Z 139.098,A -85,B 0,C 180,E1 -13269.423,E2 -13269.423} C_VEL
LIN {X 0,Y 354.788,Z 139.099,A -85,B 0,C 180,E1 -13272.867,E2 -13272.867} C_VEL
LIN {X 0,Y 354.766,Z 139.105,A -85,B 0,C 180,E1 -13276.103,E2 -13276.103} C_VEL
LIN {X 0,Y 354.787,Z 139.103,A -85,B 0,C 180,E1 -13279.179,E2 -13279.179} C_VEL
LIN {X 0,Y 354.806,Z 139.098,A -85,B 0,C 180,E1 -13282.402,E2 -13282.402} C_VEL
LIN {X 0,Y 354.811,Z 139.1,A -85,B 0,C 180,E1 -13284.941,E2 -13284.941} C_VEL
LIN {X 0,Y 354.792,Z 139.1,A -85,B 0,C 180,E1 -13288.405,E2 -13288.405} C_VEL
LIN {X 0,Y 354.848,Z 139.094,A -85,B 0,C 180,E1 -13291.619,E2 -13291.619} C_VEL
LIN {X 0,Y 354.898,Z 139.086,A -85,B 0,C 180,E1 -13294.172,E2 -13294.172} C_VEL
LIN {X 0,Y 354.833,Z 139.095,A -85,B 0,C 180,E1 -13297.894,E2 -13297.894} C_VEL
LIN {X 0,Y 354.921,Z 139.083,A -85,B 0,C 180,E1 -13301.891,E2 -13301.891} C_VEL
LIN {X 0,Y 354.942,Z 139.083,A -85,B 0,C 180,E1 -13305.981,E2 -13305.981} C_VEL
LIN {X 0,Y 354.981,Z 139.077,A -85,B 0,C 180,E1 -13309.736,E2 -13309.736} C_VEL
LIN {X 0,Y 355.113,Z 139.062,A -85,B 0,C 180,E1 -13312.037,E2 -13312.037} C_VEL
LIN {X 0,Y 355.091,Z 139.067,A -85,B 0,C 180,E1 -13314.321,E2 -13314.321} C_VEL
LIN {X 0,Y 355.244,Z 139.046,A -85,B 0,C 180,E1 -13317.732,E2 -13317.732} C_VEL
LIN {X 0,Y 355.396,Z 139.029,A -85,B 0,C 180,E1 -13320,E2 -13320} C_VEL
LIN {X 0,Y 355.242,Z 139.046,A -85,B 0,C 180,E1 -13322.268,E2 -13322.268} C_VEL
LIN {X 0,Y 355.14,Z 139.057,A -85,B 0,C 180,E1 -13326.819,E2 -13326.819} C_VEL
LIN {X 0,Y 355.013,Z 139.073,A -85,B 0,C 180,E1 -13329.112,E2 -13329.112} C_VEL
LIN {X 0,Y 354.919,Z 139.084,A -85,B 0,C 180,E1 -13332.581,E2 -13332.581} C_VEL
LIN {X 0,Y 354.888,Z 139.088,A -85,B 0,C 180,E1 -13336.096,E2 -13336.096} C_VEL
LIN {X 0,Y 354.899,Z 139.086,A -85,B 0,C 180,E1 -13338.472,E2 -13338.472} C_VEL
LIN {X 0,Y 354.833,Z 139.095,A -85,B 0,C 180,E1 -13342.106,E2 -13342.106} C_VEL
LIN {X 0,Y 354.897,Z 139.087,A -85,B 0,C 180,E1 -13345.827,E2 -13345.827} C_VEL
LIN {X 0,Y 354.852,Z 139.092,A -85,B 0,C 180,E1 -13349.679,E2 -13349.679} C_VEL
LIN {X 0,Y 354.804,Z 139.098,A -85,B 0,C 180,E1 -13353.702,E2 -13353.702} C_VEL
LIN {X 0,Y 354.796,Z 139.104,A -85,B 0,C 180,E1 -13356.46,E2 -13356.46} C_VEL
LIN {X 0,Y 354.822,Z 139.096,A -85,B 0,C 180,E1 -13359.424,E2 -13359.424} C_VEL
LIN {X 0,Y 354.786,Z 139.1,A -85,B 0,C 180,E1 -13362.867,E2 -13362.867} C_VEL
LIN {X 0,Y 354.765,Z 139.107,A -85,B 0,C 180,E1 -13366.104,E2 -13366.104} C_VEL
LIN {X 0,Y 354.786,Z 139.101,A -85,B 0,C 180,E1 -13369.179,E2 -13369.179} C_VEL
LIN {X 0,Y 354.806,Z 139.1,A -85,B 0,C 180,E1 -13372.403,E2 -13372.403} C_VEL
LIN {X 0,Y 354.811,Z 139.098,A -85,B 0,C 180,E1 -13374.941,E2 -13374.941} C_VEL
LIN {X 0,Y 354.792,Z 139.101,A -85,B 0,C 180,E1 -13378.405,E2 -13378.405} C_VEL
LIN {X 0,Y 354.85,Z 139.095,A -85,B 0,C 180,E1 -13381.619,E2 -13381.619} C_VEL
LIN {X 0,Y 354.946,Z 139.234,A -85,B 0,C 180,E1 -13384.019,E2 -13384.019} C_VEL
LIN {X 0,Y 356.826,Z 149.978,A -85,B 0,C 180,E1 -13387.347,E2 -13387.347} C_VEL
LIN {X 0,Y 356.589,Z 155.449,A -85,B 0,C 180,E1 -13388.919,E2 -13388.919} C_VEL
LIN {X 0,Y 355.571,Z 167.396,A -85,B 0,C 180,E1 -13392.234,E2 -13392.234} C_VEL
LIN {X 0,Y 356.252,Z 171.628,A -85,B 0,C 180,E1 -13392.417,E2 -13392.417} C_VEL
LIN {X 0,Y 359.75,Z 196.412,A -85,B 0,C 180,E1 -13393.099,E2 -13393.099} C_VEL
LIN {X 0,Y 359.132,Z 244.136,A -85,B 0,C 180,E1 -13394.076,E2 -13394.076} C_VEL
LIN {X 0,Y 358.72,Z 253.692,A -85,B 0,C 180,E1 -13394.409,E2 -13394.409} C_VEL
LIN {X 0,Y 358.184,Z 263.708,A -85,B 0,C 180,E1 -13394.931,E2 -13394.931} C_VEL
LIN {X 0,Y 357.367,Z 275.085,A -85,B 0,C 180,E1 -13395.77,E2 -13395.77} C_VEL
LIN {X 0,Y 356.67,Z 283.661,A -85,B 0,C 180,E1 -13396.613,E2 -13396.613} C_VEL
LIN {X 0,Y 355.939,Z 291.73,A -85,B 0,C 180,E1 -13397.601,E2 -13397.601} C_VEL
LIN {X 0,Y 355.326,Z 298.397,A -85,B 0,C 180,E1 -13398.593,E2 -13398.593} C_VEL
LIN {X 0,Y 354.724,Z 304.726,A -85,B 0,C 180,E1 -13399.729,E2 -13399.729} C_VEL
LIN {X 0,Y 354.244,Z 309.985,A -85,B 0,C 180,E1 -13400.868,E2 -13400.868} C_VEL
LIN {X 0,Y 353.864,Z 314.371,A -85,B 0,C 180,E1 -13402.009,E2 -13402.009} C_VEL
LIN {X 0,Y 353.475,Z 319.715,A -85,B 0,C 180,E1 -13403.787,E2 -13403.787} C_VEL
LIN {X 0,Y 353.343,Z 323.342,A -85,B 0,C 180,E1 -13405.437,E2 -13405.437} C_VEL
LIN {X 0,Y 353.226,Z 325.086,A -85,B 0,C 180,E1 -13406.578,E2 -13406.578} C_VEL
LIN {X 0,Y 353.151,Z 326.335,A -85,B 0,C 180,E1 -13407.719,E2 -13407.719} C_VEL
LIN {X 0,Y 353.152,Z 327.113,A -85,B 0,C 180,E1 -13408.86,E2 -13408.86} C_VEL
LIN {X 0,Y 353.19,Z 327.407,A -85,B 0,C 180,E1 -13410,E2 -13410} C_VEL
LIN {X 0,Y 353.152,Z 327.108,A -85,B 0,C 180,E1 -13411.141,E2 -13411.141} C_VEL
LIN {X 0,Y 353.151,Z 326.322,A -85,B 0,C 180,E1 -13412.281,E2 -13412.281} C_VEL
LIN {X 0,Y 353.226,Z 325.064,A -85,B 0,C 180,E1 -13413.422,E2 -13413.422} C_VEL
LIN {X 0,Y 353.352,Z 322.155,A -85,B 0,C 180,E1 -13415.135,E2 -13415.135} C_VEL
LIN {X 0,Y 353.475,Z 319.676,A -85,B 0,C 180,E1 -13416.213,E2 -13416.213} C_VEL
LIN {X 0,Y 353.715,Z 316.235,A -85,B 0,C 180,E1 -13417.421,E2 -13417.421} C_VEL
LIN {X 0,Y 354.107,Z 311.092,A -85,B 0,C 180,E1 -13418.848,E2 -13418.848} C_VEL
LIN {X 0,Y 354.619,Z 306.067,A -85,B 0,C 180,E1 -13419.986,E2 -13419.986} C_VEL
LIN {X 0,Y 355.145,Z 300.013,A -85,B 0,C 180,E1 -13421.125,E2 -13421.125} C_VEL
LIN {X 0,Y 355.844,Z 292.647,A -85,B 0,C 180,E1 -13422.258,E2 -13422.258} C_VEL
LIN {X 0,Y 356.526,Z 284.758,A -85,B 0,C 180,E1 -13423.248,E2 -13423.248} C_VEL
LIN {X 0,Y 357.256,Z 276.422,A -85,B 0,C 180,E1 -13424.09,E2 -13424.09} C_VEL
LIN {X 0,Y 358.011,Z 265.768,A -85,B 0,C 180,E1 -13424.931,E2 -13424.931} C_VEL
LIN {X 0,Y 358.625,Z 254.154,A -85,B 0,C 180,E1 -13425.559,E2 -13425.559} C_VEL
LIN {X 0,Y 359.084,Z 244.41,A -85,B 0,C 180,E1 -13425.903,E2 -13425.903} C_VEL
LIN {X 0,Y 359.56,Z 193.854,A -85,B 0,C 180,E1 -13426.946,E2 -13426.946} C_VEL
LIN {X 0,Y 355.635,Z 167.99,A -85,B 0,C 180,E1 -13427.691,E2 -13427.691} C_VEL
LIN {X 0,Y 355.589,Z 166.971,A -85,B 0,C 180,E1 -13427.839,E2 -13427.839} C_VEL
LIN {X 0,Y 356.769,Z 153.291,A -85,B 0,C 180,E1 -13431.676,E2 -13431.676} C_VEL
LIN {X 0,Y 356.816,Z 149.94,A -85,B 0,C 180,E1 -13432.646,E2 -13432.646} C_VEL
LIN {X 0,Y 354.948,Z 139.199,A -85,B 0,C 180,E1 -13435.981,E2 -13435.981} C_VEL
LIN {X 0,Y 354.854,Z 139.092,A -85,B 0,C 180,E1 -13439.679,E2 -13439.679} C_VEL
LIN {X 0,Y 354.807,Z 139.099,A -85,B 0,C 180,E1 -13443.702,E2 -13443.702} C_VEL
LIN {X 0,Y 354.799,Z 139.101,A -85,B 0,C 180,E1 -13446.46,E2 -13446.46} C_VEL
LIN {X 0,Y 354.825,Z 139.096,A -85,B 0,C 180,E1 -13449.424,E2 -13449.424} C_VEL
LIN {X 0,Y 354.789,Z 139.1,A -85,B 0,C 180,E1 -13452.867,E2 -13452.867} C_VEL
LIN {X 0,Y 354.768,Z 139.103,A -85,B 0,C 180,E1 -13456.104,E2 -13456.104} C_VEL
LIN {X 0,Y 354.788,Z 139.102,A -85,B 0,C 180,E1 -13459.179,E2 -13459.179} C_VEL
LIN {X 0,Y 354.807,Z 139.098,A -85,B 0,C 180,E1 -13462.403,E2 -13462.403} C_VEL
LIN {X 0,Y 354.813,Z 139.099,A -85,B 0,C 180,E1 -13464.941,E2 -13464.941} C_VEL
LIN {X 0,Y 354.794,Z 139.1,A -85,B 0,C 180,E1 -13468.405,E2 -13468.405} C_VEL
LIN {X 0,Y 354.852,Z 139.093,A -85,B 0,C 180,E1 -13471.619,E2 -13471.619} C_VEL
LIN {X 0,Y 354.9,Z 139.086,A -85,B 0,C 180,E1 -13474.173,E2 -13474.173} C_VEL
LIN {X 0,Y 354.836,Z 139.094,A -85,B 0,C 180,E1 -13477.894,E2 -13477.894} C_VEL
LIN {X 0,Y 354.924,Z 139.083,A -85,B 0,C 180,E1 -13481.892,E2 -13481.892} C_VEL
LIN {X 0,Y 354.944,Z 139.082,A -85,B 0,C 180,E1 -13485.981,E2 -13485.981} C_VEL
LIN {X 0,Y 354.98,Z 139.076,A -85,B 0,C 180,E1 -13489.736,E2 -13489.736} C_VEL
LIN {X 0,Y 355.126,Z 139.058,A -85,B 0,C 180,E1 -13493.181,E2 -13493.181} C_VEL
LIN {X 0,Y 355.245,Z 139.045,A -85,B 0,C 180,E1 -13497.733,E2 -13497.733} C_VEL
LIN {X 0,Y 355.377,Z 139.031,A -85,B 0,C 180,E1 -13500,E2 -13500} C_VEL
LIN {X 0,Y 355.245,Z 139.047,A -85,B 0,C 180,E1 -13502.268,E2 -13502.268} C_VEL
LIN {X 0,Y 355.14,Z 139.056,A -85,B 0,C 180,E1 -13506.819,E2 -13506.819} C_VEL
LIN {X 0,Y 355.019,Z 139.072,A -85,B 0,C 180,E1 -13509.112,E2 -13509.112} C_VEL
LIN {X 0,Y 354.928,Z 139.083,A -85,B 0,C 180,E1 -13512.581,E2 -13512.581} C_VEL
LIN {X 0,Y 354.892,Z 139.088,A -85,B 0,C 180,E1 -13516.096,E2 -13516.096} C_VEL
LIN {X 0,Y 354.903,Z 139.085,A -85,B 0,C 180,E1 -13518.472,E2 -13518.472} C_VEL
LIN {X 0,Y 354.836,Z 139.094,A -85,B 0,C 180,E1 -13522.106,E2 -13522.106} C_VEL
LIN {X 0,Y 354.901,Z 139.086,A -85,B 0,C 180,E1 -13525.827,E2 -13525.827} C_VEL
LIN {X 0,Y 354.855,Z 139.092,A -85,B 0,C 180,E1 -13529.679,E2 -13529.679} C_VEL
LIN {X 0,Y 354.808,Z 139.097,A -85,B 0,C 180,E1 -13533.702,E2 -13533.702} C_VEL
LIN {X 0,Y 354.799,Z 139.102,A -85,B 0,C 180,E1 -13536.459,E2 -13536.459} C_VEL
LIN {X 0,Y 354.826,Z 139.095,A -85,B 0,C 180,E1 -13539.424,E2 -13539.424} C_VEL
LIN {X 0,Y 354.789,Z 139.102,A -85,B 0,C 180,E1 -13542.867,E2 -13542.867} C_VEL
LIN {X 0,Y 354.769,Z 139.106,A -85,B 0,C 180,E1 -13546.104,E2 -13546.104} C_VEL
LIN {X 0,Y 354.79,Z 139.1,A -85,B 0,C 180,E1 -13549.179,E2 -13549.179} C_VEL
LIN {X 0,Y 354.81,Z 139.1,A -85,B 0,C 180,E1 -13552.402,E2 -13552.402} C_VEL
LIN {X 0,Y 354.814,Z 139.096,A -85,B 0,C 180,E1 -13554.941,E2 -13554.941} C_VEL
LIN {X 0,Y 354.795,Z 139.101,A -85,B 0,C 180,E1 -13558.405,E2 -13558.405} C_VEL
LIN {X 0,Y 354.853,Z 139.097,A -85,B 0,C 180,E1 -13561.619,E2 -13561.619} C_VEL
LIN {X 0,Y 354.901,Z 139.088,A -85,B 0,C 180,E1 -13564.172,E2 -13564.172} C_VEL
LIN {X 0,Y 354.902,Z 139.286,A -85,B 0,C 180,E1 -13567.285,E2 -13567.285} C_VEL
LIN {X 0,Y 355.943,Z 145.038,A -85,B 0,C 180,E1 -13569.182,E2 -13569.182} C_VEL
LIN {X 0,Y 356.069,Z 150.792,A -85,B 0,C 180,E1 -13570.967,E2 -13570.967} C_VEL
LIN {X 0,Y 355.818,Z 155.315,A -85,B 0,C 180,E1 -13572.295,E2 -13572.295} C_VEL
LIN {X 0,Y 356.09,Z 157.115,A -85,B 0,C 180,E1 -13572.424,E2 -13572.424} C_VEL
LIN {X 0,Y 359.907,Z 179.121,A -85,B 0,C 180,E1 -13573.069,E2 -13573.069} C_VEL
LIN {X 0,Y 359.174,Z 231.604,A -85,B 0,C 180,E1 -13574.137,E2 -13574.137} C_VEL
LIN {X 0,Y 358.844,Z 241.451,A -85,B 0,C 180,E1 -13574.487,E2 -13574.487} C_VEL
LIN {X 0,Y 358.387,Z 252.572,A -85,B 0,C 180,E1 -13575.085,E2 -13575.085} C_VEL
LIN {X 0,Y 357.664,Z 263.411,A -85,B 0,C 180,E1 -13575.926,E2 -13575.926} C_VEL
LIN {X 0,Y 356.947,Z 271.811,A -85,B 0,C 180,E1 -13576.768,E2 -13576.768} C_VEL
LIN {X 0,Y 356.302,Z 279.739,A -85,B 0,C 180,E1 -13577.758,E2 -13577.758} C_VEL
LIN {X 0,Y 355.796,Z 285.432,A -85,B 0,C 180,E1 -13578.607,E2 -13578.607} C_VEL
LIN {X 0,Y 355.159,Z 291.788,A -85,B 0,C 180,E1 -13579.741,E2 -13579.741} C_VEL
LIN {X 0,Y 354.593,Z 297.071,A -85,B 0,C 180,E1 -13580.876,E2 -13580.876} C_VEL
LIN {X 0,Y 354.265,Z 301.479,A -85,B 0,C 180,E1 -13582.017,E2 -13582.017} C_VEL
LIN {X 0,Y 353.962,Z 305.151,A -85,B 0,C 180,E1 -13583.158,E2 -13583.158} C_VEL
LIN {X 0,Y 353.724,Z 308.149,A -85,B 0,C 180,E1 -13584.298,E2 -13584.298} C_VEL
LIN {X 0,Y 353.53,Z 310.472,A -85,B 0,C 180,E1 -13585.439,E2 -13585.439} C_VEL
LIN {X 0,Y 353.327,Z 312.24,A -85,B 0,C 180,E1 -13586.579,E2 -13586.579} C_VEL
LIN {X 0,Y 353.22,Z 313.515,A -85,B 0,C 180,E1 -13587.719,E2 -13587.719} C_VEL
LIN {X 0,Y 353.183,Z 314.319,A -85,B 0,C 180,E1 -13588.86,E2 -13588.86} C_VEL
LIN {X 0,Y 353.194,Z 314.625,A -85,B 0,C 180,E1 -13590,E2 -13590} C_VEL
LIN {X 0,Y 353.183,Z 314.349,A -85,B 0,C 180,E1 -13591.14,E2 -13591.14} C_VEL
LIN {X 0,Y 353.219,Z 313.604,A -85,B 0,C 180,E1 -13592.28,E2 -13592.28} C_VEL
LIN {X 0,Y 353.323,Z 312.39,A -85,B 0,C 180,E1 -13593.421,E2 -13593.421} C_VEL
LIN {X 0,Y 353.616,Z 309.537,A -85,B 0,C 180,E1 -13595.131,E2 -13595.131} C_VEL
LIN {X 0,Y 353.778,Z 306.849,A -85,B 0,C 180,E1 -13596.308,E2 -13596.308} C_VEL
LIN {X 0,Y 354.233,Z 301.834,A -85,B 0,C 180,E1 -13597.983,E2 -13597.983} C_VEL
LIN {X 0,Y 354.695,Z 296.337,A -85,B 0,C 180,E1 -13599.408,E2 -13599.408} C_VEL
LIN {X 0,Y 355.425,Z 289.43,A -85,B 0,C 180,E1 -13600.827,E2 -13600.827} C_VEL
LIN {X 0,Y 356.166,Z 281.499,A -85,B 0,C 180,E1 -13602.102,E2 -13602.102} C_VEL
LIN {X 0,Y 356.875,Z 273.934,A -85,B 0,C 180,E1 -13603.089,E2 -13603.089} C_VEL
LIN {X 0,Y 357.54,Z 266.006,A -85,B 0,C 180,E1 -13603.933,E2 -13603.933} C_VEL
LIN {X 0,Y 358.053,Z 257.818,A -85,B 0,C 180,E1 -13604.638,E2 -13604.638} C_VEL
LIN {X 0,Y 358.593,Z 249.519,A -85,B 0,C 180,E1 -13605.196,E2 -13605.196} C_VEL
LIN {X 0,Y 358.961,Z 240.553,A -85,B 0,C 180,E1 -13605.653,E2 -13605.653} C_VEL
LIN {X 0,Y 359.257,Z 231.06,A -85,B 0,C 180,E1 -13605.98,E2 -13605.98} C_VEL
LIN {X 0,Y 359.756,Z 177.233,A -85,B 0,C 180,E1 -13607.083,E2 -13607.083} C_VEL
LIN {X 0,Y 355.853,Z 155.885,A -85,B 0,C 180,E1 -13607.744,E2 -13607.744} C_VEL
LIN {X 0,Y 355.858,Z 154.656,A -85,B 0,C 180,E1 -13607.974,E2 -13607.974} C_VEL
LIN {X 0,Y 356.123,Z 149.889,A -85,B 0,C 180,E1 -13609.416,E2 -13609.416} C_VEL
LIN {X 0,Y 355.467,Z 148.199,A -85,B 0,C 180,E1 -13609.978,E2 -13609.978} C_VEL
LIN {X 0,Y 352.465,Z 145.947,A -85,B 0,C 180,E1 -13610.876,E2 -13610.876} C_VEL
LIN {X 0,Y 349.22,Z 143.764,A -85,B 0,C 180,E1 -13611.791,E2 -13611.791} C_VEL
LIN {X 0,Y 348.23,Z 142.157,A -85,B 0,C 180,E1 -13612.377,E2 -13612.377} C_VEL
LIN {X 0,Y 347.846,Z 140.079,A -85,B 0,C 180,E1 -13613.124,E2 -13613.124} C_VEL
LIN {X 0,Y 347.852,Z 139.964,A -85,B 0,C 180,E1 -13617.255,E2 -13617.255} C_VEL
LIN {X 0,Y 347.764,Z 139.98,A -85,B 0,C 180,E1 -13620.346,E2 -13620.346} C_VEL
LIN {X 0,Y 347.744,Z 139.978,A -85,B 0,C 180,E1 -13624.463,E2 -13624.463} C_VEL
LIN {X 0,Y 347.774,Z 139.98,A -85,B 0,C 180,E1 -13627.988,E2 -13627.988} C_VEL
LIN {X 0,Y 347.75,Z 139.979,A -85,B 0,C 180,E1 -13631.83,E2 -13631.83} C_VEL
LIN {X 0,Y 347.705,Z 139.982,A -85,B 0,C 180,E1 -13635.026,E2 -13635.026} C_VEL
LIN {X 0,Y 347.749,Z 139.977,A -85,B 0,C 180,E1 -13638.397,E2 -13638.397} C_VEL
LIN {X 0,Y 347.772,Z 139.976,A -85,B 0,C 180,E1 -13642.011,E2 -13642.011} C_VEL
LIN {X 0,Y 347.743,Z 139.98,A -85,B 0,C 180,E1 -13645.536,E2 -13645.536} C_VEL
LIN {X 0,Y 347.763,Z 139.977,A -85,B 0,C 180,E1 -13649.653,E2 -13649.653} C_VEL
LIN {X 0,Y 347.85,Z 139.967,A -85,B 0,C 180,E1 -13652.745,E2 -13652.745} C_VEL
LIN {X 0,Y 347.787,Z 139.973,A -85,B 0,C 180,E1 -13656.162,E2 -13656.162} C_VEL
LIN {X 0,Y 347.811,Z 139.969,A -85,B 0,C 180,E1 -13659.909,E2 -13659.909} C_VEL
LIN {X 0,Y 347.865,Z 139.964,A -85,B 0,C 180,E1 -13662.359,E2 -13662.359} C_VEL
LIN {X 0,Y 347.896,Z 139.96,A -85,B 0,C 180,E1 -13665.971,E2 -13665.971} C_VEL
LIN {X 0,Y 347.932,Z 139.954,A -85,B 0,C 180,E1 -13669.526,E2 -13669.526} C_VEL
LIN {X 0,Y 348.073,Z 139.937,A -85,B 0,C 180,E1 -13671.875,E2 -13671.875} C_VEL
LIN {X 0,Y 348.066,Z 139.943,A -85,B 0,C 180,E1 -13674.206,E2 -13674.206} C_VEL
LIN {X 0,Y 348.207,Z 139.923,A -85,B 0,C 180,E1 -13677.686,E2 -13677.686} C_VEL
LIN {X 0,Y 348.345,Z 139.906,A -85,B 0,C 180,E1 -13680,E2 -13680} C_VEL
LIN {X 0,Y 348.205,Z 139.922,A -85,B 0,C 180,E1 -13682.313,E2 -13682.313} C_VEL
LIN {X 0,Y 348.107,Z 139.933,A -85,B 0,C 180,E1 -13686.957,E2 -13686.957} C_VEL
LIN {X 0,Y 347.966,Z 139.952,A -85,B 0,C 180,E1 -13689.298,E2 -13689.298} C_VEL
LIN {X 0,Y 347.888,Z 139.96,A -85,B 0,C 180,E1 -13692.839,E2 -13692.839} C_VEL
LIN {X 0,Y 347.837,Z 139.966,A -85,B 0,C 180,E1 -13696.431,E2 -13696.431} C_VEL
LIN {X 0,Y 347.849,Z 139.966,A -85,B 0,C 180,E1 -13698.86,E2 -13698.86} C_VEL
LIN {X 0,Y 347.772,Z 139.975,A -85,B 0,C 180,E1 -13702.579,E2 -13702.579} C_VEL
LIN {X 0,Y 347.811,Z 139.974,A -85,B 0,C 180,E1 -13705.108,E2 -13705.108} C_VEL
LIN {X 0,Y 347.809,Z 139.969,A -85,B 0,C 180,E1 -13707.694,E2 -13707.694} C_VEL
LIN {X 0,Y 347.762,Z 139.977,A -85,B 0,C 180,E1 -13710.347,E2 -13710.347} C_VEL
LIN {X 0,Y 347.742,Z 139.981,A -85,B 0,C 180,E1 -13714.464,E2 -13714.464} C_VEL
LIN {X 0,Y 347.771,Z 139.976,A -85,B 0,C 180,E1 -13717.989,E2 -13717.989} C_VEL
LIN {X 0,Y 347.749,Z 139.977,A -85,B 0,C 180,E1 -13721.83,E2 -13721.83} C_VEL
LIN {X 0,Y 347.704,Z 139.982,A -85,B 0,C 180,E1 -13725.027,E2 -13725.027} C_VEL
LIN {X 0,Y 347.749,Z 139.98,A -85,B 0,C 180,E1 -13728.397,E2 -13728.397} C_VEL
LIN {X 0,Y 347.772,Z 139.978,A -85,B 0,C 180,E1 -13732.012,E2 -13732.012} C_VEL
LIN {X 0,Y 347.743,Z 139.981,A -85,B 0,C 180,E1 -13735.536,E2 -13735.536} C_VEL
LIN {X 0,Y 347.763,Z 139.981,A -85,B 0,C 180,E1 -13739.654,E2 -13739.654} C_VEL
LIN {X 0,Y 347.887,Z 140.012,A -85,B 0,C 180,E1 -13743.693,E2 -13743.693} C_VEL
LIN {X 0,Y 349.696,Z 150.08,A -85,B 0,C 180,E1 -13746.928,E2 -13746.928} C_VEL
LIN {X 0,Y 349.903,Z 153.229,A -85,B 0,C 180,E1 -13747.877,E2 -13747.877} C_VEL
LIN {X 0,Y 348.608,Z 167.11,A -85,B 0,C 180,E1 -13751.84,E2 -13751.84} C_VEL
LIN {X 0,Y 348.928,Z 169.347,A -85,B 0,C 180,E1 -13751.99,E2 -13751.99} C_VEL
LIN {X 0,Y 352.931,Z 195.916,A -85,B 0,C 180,E1 -13752.755,E2 -13752.755} C_VEL
LIN {X 0,Y 352.322,Z 244.074,A -85,B 0,C 180,E1 -13753.761,E2 -13753.761} C_VEL
LIN {X 0,Y 351.88,Z 253.573,A -85,B 0,C 180,E1 -13754.098,E2 -13754.098} C_VEL
LIN {X 0,Y 351.349,Z 263.587,A -85,B 0,C 180,E1 -13754.631,E2 -13754.631} C_VEL
LIN {X 0,Y 350.493,Z 274.961,A -85,B 0,C 180,E1 -13755.485,E2 -13755.485} C_VEL
LIN {X 0,Y 349.782,Z 283.536,A -85,B 0,C 180,E1 -13756.345,E2 -13756.345} C_VEL
LIN {X 0,Y 348.977,Z 291.604,A -85,B 0,C 180,E1 -13757.349,E2 -13757.349} C_VEL
LIN {X 0,Y 348.37,Z 298.271,A -85,B 0,C 180,E1 -13758.362,E2 -13758.362} C_VEL
LIN {X 0,Y 347.736,Z 304.599,A -85,B 0,C 180,E1 -13759.52,E2 -13759.52} C_VEL
LIN {X 0,Y 347.225,Z 309.858,A -85,B 0,C 180,E1 -13760.682,E2 -13760.682} C_VEL
LIN {X 0,Y 346.822,Z 314.243,A -85,B 0,C 180,E1 -13761.846,E2 -13761.846} C_VEL
LIN {X 0,Y 346.424,Z 319.417,A -85,B 0,C 180,E1 -13763.594,E2 -13763.594} C_VEL
LIN {X 0,Y 346.259,Z 323.214,A -85,B 0,C 180,E1 -13765.343,E2 -13765.343} C_VEL
LIN {X 0,Y 346.153,Z 324.959,A -85,B 0,C 180,E1 -13766.508,E2 -13766.508} C_VEL
LIN {X 0,Y 346.065,Z 326.207,A -85,B 0,C 180,E1 -13767.672,E2 -13767.672} C_VEL
LIN {X 0,Y 346.055,Z 326.984,A -85,B 0,C 180,E1 -13768.837,E2 -13768.837} C_VEL
LIN {X 0,Y 346.092,Z 327.278,A -85,B 0,C 180,E1 -13770,E2 -13770} C_VEL
LIN {X 0,Y 346.055,Z 326.979,A -85,B 0,C 180,E1 -13771.164,E2 -13771.164} C_VEL
LIN {X 0,Y 346.065,Z 326.193,A -85,B 0,C 180,E1 -13772.328,E2 -13772.328} C_VEL
LIN {X 0,Y 346.153,Z 324.935,A -85,B 0,C 180,E1 -13773.492,E2 -13773.492} C_VEL
LIN {X 0,Y 346.259,Z 322.025,A -85,B 0,C 180,E1 -13775.241,E2 -13775.241} C_VEL
LIN {X 0,Y 346.469,Z 318.876,A -85,B 0,C 180,E1 -13776.597,E2 -13776.597} C_VEL
LIN {X 0,Y 346.85,Z 313.223,A -85,B 0,C 180,E1 -13778.448,E2 -13778.448} C_VEL
LIN {X 0,Y 347.478,Z 307.352,A -85,B 0,C 180,E1 -13779.9,E2 -13779.9} C_VEL
LIN {X 0,Y 348.169,Z 299.882,A -85,B 0,C 180,E1 -13781.351,E2 -13781.351} C_VEL
LIN {X 0,Y 348.888,Z 292.516,A -85,B 0,C 180,E1 -13782.507,E2 -13782.507} C_VEL
LIN {X 0,Y 349.622,Z 284.627,A -85,B 0,C 180,E1 -13783.514,E2 -13783.514} C_VEL
LIN {X 0,Y 350.369,Z 276.289,A -85,B 0,C 180,E1 -13784.373,E2 -13784.373} C_VEL
LIN {X 0,Y 351.153,Z 265.633,A -85,B 0,C 180,E1 -13785.23,E2 -13785.23} C_VEL
LIN {X 0,Y 351.807,Z 254.017,A -85,B 0,C 180,E1 -13785.869,E2 -13785.869} C_VEL
LIN {X 0,Y 352.28,Z 244.267,A -85,B 0,C 180,E1 -13786.219,E2 -13786.219} C_VEL
LIN {X 0,Y 352.776,Z 194.742,A -85,B 0,C 180,E1 -13787.261,E2 -13787.261} C_VEL
LIN {X 0,Y 348.731,Z 168.213,A -85,B 0,C 180,E1 -13788.04,E2 -13788.04} C_VEL
LIN {X 0,Y 348.609,Z 167.042,A -85,B 0,C 180,E1 -13788.161,E2 -13788.161} C_VEL
LIN {X 0,Y 349.799,Z 154.209,A -85,B 0,C 180,E1 -13791.82,E2 -13791.82} C_VEL
LIN {X 0,Y 349.657,Z 150.01,A -85,B 0,C 180,E1 -13793.075,E2 -13793.075} C_VEL
LIN {X 0,Y 347.908,Z 140.039,A -85,B 0,C 180,E1 -13796.265,E2 -13796.265} C_VEL
LIN {X 0,Y 347.764,Z 139.98,A -85,B 0,C 180,E1 -13800.347,E2 -13800.347} C_VEL
LIN {X 0,Y 347.745,Z 139.981,A -85,B 0,C 180,E1 -13804.464,E2 -13804.464} C_VEL
LIN {X 0,Y 347.774,Z 139.978,A -85,B 0,C 180,E1 -13807.989,E2 -13807.989} C_VEL
LIN {X 0,Y 347.751,Z 139.982,A -85,B 0,C 180,E1 -13811.83,E2 -13811.83} C_VEL
LIN {X 0,Y 347.706,Z 139.981,A -85,B 0,C 180,E1 -13815.027,E2 -13815.027} C_VEL
LIN {X 0,Y 347.751,Z 139.976,A -85,B 0,C 180,E1 -13818.397,E2 -13818.397} C_VEL
LIN {X 0,Y 347.774,Z 139.976,A -85,B 0,C 180,E1 -13822.012,E2 -13822.012} C_VEL
LIN {X 0,Y 347.745,Z 139.981,A -85,B 0,C 180,E1 -13825.536,E2 -13825.536} C_VEL
LIN {X 0,Y 347.765,Z 139.977,A -85,B 0,C 180,E1 -13829.654,E2 -13829.654} C_VEL
LIN {X 0,Y 347.853,Z 139.965,A -85,B 0,C 180,E1 -13832.745,E2 -13832.745} C_VEL
LIN {X 0,Y 347.79,Z 139.972,A -85,B 0,C 180,E1 -13836.162,E2 -13836.162} C_VEL
LIN {X 0,Y 347.814,Z 139.968,A -85,B 0,C 180,E1 -13839.91,E2 -13839.91} C_VEL
LIN {X 0,Y 347.867,Z 139.964,A -85,B 0,C 180,E1 -13842.359,E2 -13842.359} C_VEL
LIN {X 0,Y 347.899,Z 139.959,A -85,B 0,C 180,E1 -13845.971,E2 -13845.971} C_VEL
LIN {X 0,Y 347.93,Z 139.952,A -85,B 0,C 180,E1 -13849.526,E2 -13849.526} C_VEL
LIN {X 0,Y 348.092,Z 139.935,A -85,B 0,C 180,E1 -13853.042,E2 -13853.042} C_VEL
LIN {X 0,Y 348.207,Z 139.921,A -85,B 0,C 180,E1 -13857.687,E2 -13857.687} C_VEL
LIN {X 0,Y 348.327,Z 139.908,A -85,B 0,C 180,E1 -13860,E2 -13860} C_VEL
LIN {X 0,Y 348.207,Z 139.923,A -85,B 0,C 180,E1 -13862.314,E2 -13862.314} C_VEL
LIN {X 0,Y 348.108,Z 139.932,A -85,B 0,C 180,E1 -13866.958,E2 -13866.958} C_VEL
LIN {X 0,Y 347.971,Z 139.949,A -85,B 0,C 180,E1 -13869.299,E2 -13869.299} C_VEL
LIN {X 0,Y 347.896,Z 139.959,A -85,B 0,C 180,E1 -13872.839,E2 -13872.839} C_VEL
LIN {X 0,Y 347.841,Z 139.965,A -85,B 0,C 180,E1 -13876.431,E2 -13876.431} C_VEL
LIN {X 0,Y 347.853,Z 139.964,A -85,B 0,C 180,E1 -13878.861,E2 -13878.861} C_VEL
LIN {X 0,Y 347.776,Z 139.975,A -85,B 0,C 180,E1 -13882.579,E2 -13882.579} C_VEL
LIN {X 0,Y 347.815,Z 139.974,A -85,B 0,C 180,E1 -13885.108,E2 -13885.108} C_VEL
LIN {X 0,Y 347.811,Z 139.969,A -85,B 0,C 180,E1 -13887.694,E2 -13887.694} C_VEL
LIN {X 0,Y 347.766,Z 139.976,A -85,B 0,C 180,E1 -13890.346,E2 -13890.346} C_VEL
LIN {X 0,Y 347.746,Z 139.979,A -85,B 0,C 180,E1 -13894.464,E2 -13894.464} C_VEL
LIN {X 0,Y 347.775,Z 139.975,A -85,B 0,C 180,E1 -13897.989,E2 -13897.989} C_VEL
LIN {X 0,Y 347.752,Z 139.977,A -85,B 0,C 180,E1 -13901.83,E2 -13901.83} C_VEL
LIN {X 0,Y 347.707,Z 139.982,A -85,B 0,C 180,E1 -13905.027,E2 -13905.027} C_VEL
LIN {X 0,Y 347.752,Z 139.98,A -85,B 0,C 180,E1 -13908.397,E2 -13908.397} C_VEL
LIN {X 0,Y 347.776,Z 139.979,A -85,B 0,C 180,E1 -13912.011,E2 -13912.011} C_VEL
LIN {X 0,Y 347.746,Z 139.977,A -85,B 0,C 180,E1 -13915.536,E2 -13915.536} C_VEL
LIN {X 0,Y 347.766,Z 139.979,A -85,B 0,C 180,E1 -13919.653,E2 -13919.653} C_VEL
LIN {X 0,Y 347.854,Z 139.964,A -85,B 0,C 180,E1 -13922.745,E2 -13922.745} C_VEL
LIN {X 0,Y 347.82,Z 139.992,A -85,B 0,C 180,E1 -13926.795,E2 -13926.795} C_VEL
LIN {X 0,Y 347.888,Z 140.33,A -85,B 0,C 180,E1 -13927.115,E2 -13927.115} C_VEL
LIN {X 0,Y 349.046,Z 147.102,A -85,B 0,C 180,E1 -13929.368,E2 -13929.368} C_VEL
LIN {X 0,Y 349.055,Z 152.957,A -85,B 0,C 180,E1 -13931.207,E2 -13931.207} C_VEL
LIN {X 0,Y 348.901,Z 155.751,A -85,B 0,C 180,E1 -13931.973,E2 -13931.973} C_VEL
LIN {X 0,Y 350.025,Z 161.765,A -85,B 0,C 180,E1 -13932.205,E2 -13932.205} C_VEL
LIN {X 0,Y 353.127,Z 179.947,A -85,B 0,C 180,E1 -13932.748,E2 -13932.748} C_VEL
LIN {X 0,Y 352.372,Z 231.75,A -85,B 0,C 180,E1 -13933.823,E2 -13933.823} C_VEL
LIN {X 0,Y 352.021,Z 241.591,A -85,B 0,C 180,E1 -13934.178,E2 -13934.178} C_VEL
LIN {X 0,Y 351.551,Z 252.708,A -85,B 0,C 180,E1 -13934.788,E2 -13934.788} C_VEL
LIN {X 0,Y 350.793,Z 263.545,A -85,B 0,C 180,E1 -13935.645,E2 -13935.645} C_VEL
LIN {X 0,Y 350.042,Z 271.944,A -85,B 0,C 180,E1 -13936.502,E2 -13936.502} C_VEL
LIN {X 0,Y 349.385,Z 279.871,A -85,B 0,C 180,E1 -13937.511,E2 -13937.511} C_VEL
LIN {X 0,Y 348.84,Z 285.563,A -85,B 0,C 180,E1 -13938.377,E2 -13938.377} C_VEL
LIN {X 0,Y 348.163,Z 291.919,A -85,B 0,C 180,E1 -13939.532,E2 -13939.532} C_VEL
LIN {X 0,Y 347.574,Z 297.202,A -85,B 0,C 180,E1 -13940.691,E2 -13940.691} C_VEL
LIN {X 0,Y 347.221,Z 301.61,A -85,B 0,C 180,E1 -13941.854,E2 -13941.854} C_VEL
LIN {X 0,Y 346.892,Z 305.47,A -85,B 0,C 180,E1 -13943.091,E2 -13943.091} C_VEL
LIN {X 0,Y 346.562,Z 309.454,A -85,B 0,C 180,E1 -13944.764,E2 -13944.764} C_VEL
LIN {X 0,Y 346.254,Z 312.369,A -85,B 0,C 180,E1 -13946.509,E2 -13946.509} C_VEL
LIN {X 0,Y 346.132,Z 313.643,A -85,B 0,C 180,E1 -13947.672,E2 -13947.672} C_VEL
LIN {X 0,Y 346.085,Z 314.447,A -85,B 0,C 180,E1 -13948.836,E2 -13948.836} C_VEL
LIN {X 0,Y 346.096,Z 314.753,A -85,B 0,C 180,E1 -13950,E2 -13950} C_VEL
LIN {X 0,Y 346.085,Z 314.477,A -85,B 0,C 180,E1 -13951.163,E2 -13951.163} C_VEL
LIN {X 0,Y 346.131,Z 313.732,A -85,B 0,C 180,E1 -13952.327,E2 -13952.327} C_VEL
LIN {X 0,Y 346.25,Z 312.518,A -85,B 0,C 180,E1 -13953.491,E2 -13953.491} C_VEL
LIN {X 0,Y 346.546,Z 309.665,A -85,B 0,C 180,E1 -13955.236,E2 -13955.236} C_VEL
LIN {X 0,Y 346.807,Z 306.053,A -85,B 0,C 180,E1 -13956.792,E2 -13956.792} C_VEL
LIN {X 0,Y 347.199,Z 301.96,A -85,B 0,C 180,E1 -13958.146,E2 -13958.146} C_VEL
LIN {X 0,Y 347.685,Z 296.464,A -85,B 0,C 180,E1 -13959.599,E2 -13959.599} C_VEL
LIN {X 0,Y 348.458,Z 289.556,A -85,B 0,C 180,E1 -13961.046,E2 -13961.046} C_VEL
LIN {X 0,Y 349.227,Z 281.624,A -85,B 0,C 180,E1 -13962.346,E2 -13962.346} C_VEL
LIN {X 0,Y 349.967,Z 274.058,A -85,B 0,C 180,E1 -13963.352,E2 -13963.352} C_VEL
LIN {X 0,Y 350.665,Z 266.129,A -85,B 0,C 180,E1 -13964.212,E2 -13964.212} C_VEL
LIN {X 0,Y 351.212,Z 257.94,A -85,B 0,C 180,E1 -13964.93,E2 -13964.93} C_VEL
LIN {X 0,Y 351.762,Z 249.639,A -85,B 0,C 180,E1 -13965.499,E2 -13965.499} C_VEL
LIN {X 0,Y 352.146,Z 240.67,A -85,B 0,C 180,E1 -13965.964,E2 -13965.964} C_VEL
LIN {X 0,Y 352.453,Z 231.3,A -85,B 0,C 180,E1 -13966.293,E2 -13966.293} C_VEL
LIN {X 0,Y 352.987,Z 178.233,A -85,B 0,C 180,E1 -13967.402,E2 -13967.402} C_VEL
LIN {X 0,Y 348.946,Z 156.013,A -85,B 0,C 180,E1 -13968.106,E2 -13968.106} C_VEL
LIN {X 0,Y 348.921,Z 154.777,A -85,B 0,C 180,E1 -13968.344,E2 -13968.344} C_VEL
LIN {X 0,Y 349.166,Z 149.401,A -85,B 0,C 180,E1 -13970.009,E2 -13970.009} C_VEL
LIN {X 0,Y 348.501,Z 143.494,A -85,B 0,C 180,E1 -13971.928,E2 -13971.928} C_VEL
LIN {X 0,Y 348.23,Z 142.157,A -85,B 0,C 180,E1 -13972.377,E2 -13972.377} C_VEL
LIN {X 0,Y 347.633,Z 140.901,A -85,B 0,C 180,E1 -13972.971,E2 -13972.971} C_VEL
LIN {X 0,Y 346.068,Z 140.275,A -85,B 0,C 180,E1 -13973.898,E2 -13973.898} C_VEL
LIN {X 0,Y 341.84,Z 140.725,A -85,B 0,C 180,E1 -13976.135,E2 -13976.135} C_VEL
LIN {X 0,Y 340.862,Z 140.836,A -85,B 0,C 180,E1 -13977.14,E2 -13977.14} C_VEL
LIN {X 0,Y 340.78,Z 140.845,A -85,B 0,C 180,E1 -13977.479,E2 -13977.479} C_VEL
LIN {X 0,Y 340.704,Z 140.855,A -85,B 0,C 180,E1 -13981.044,E2 -13981.044} C_VEL
LIN {X 0,Y 340.718,Z 140.85,A -85,B 0,C 180,E1 -13985.278,E2 -13985.278} C_VEL
LIN {X 0,Y 340.71,Z 140.856,A -85,B 0,C 180,E1 -13988.386,E2 -13988.386} C_VEL
LIN {X 0,Y 340.698,Z 140.853,A -85,B 0,C 180,E1 -13992.045,E2 -13992.045} C_VEL
LIN {X 0,Y 340.651,Z 140.863,A -85,B 0,C 180,E1 -13996.227,E2 -13996.227} C_VEL
LIN {X 0,Y 340.687,Z 140.859,A -85,B 0,C 180,E1 -13999.753,E2 -13999.753} C_VEL
LIN {X 0,Y 340.704,Z 140.86,A -85,B 0,C 180,E1 -14003.258,E2 -14003.258} C_VEL
LIN {X 0,Y 340.691,Z 140.854,A -85,B 0,C 180,E1 -14006.153,E2 -14006.153} C_VEL
LIN {X 0,Y 340.773,Z 140.847,A -85,B 0,C 180,E1 -14010.332,E2 -14010.332} C_VEL
LIN {X 0,Y 340.803,Z 140.846,A -85,B 0,C 180,E1 -14013.02,E2 -14013.02} C_VEL
LIN {X 0,Y 340.755,Z 140.849,A -85,B 0,C 180,E1 -14015.638,E2 -14015.638} C_VEL
LIN {X 0,Y 340.751,Z 140.849,A -85,B 0,C 180,E1 -14019.474,E2 -14019.474} C_VEL
LIN {X 0,Y 340.856,Z 140.833,A -85,B 0,C 180,E1 -14021.984,E2 -14021.984} C_VEL
LIN {X 0,Y 340.868,Z 140.835,A -85,B 0,C 180,E1 -14025.705,E2 -14025.705} C_VEL
LIN {X 0,Y 340.874,Z 140.832,A -85,B 0,C 180,E1 -14029.306,E2 -14029.306} C_VEL
LIN {X 0,Y 341.075,Z 140.808,A -85,B 0,C 180,E1 -14032.898,E2 -14032.898} C_VEL
LIN {X 0,Y 341.168,Z 140.799,A -85,B 0,C 180,E1 -14037.639,E2 -14037.639} C_VEL
LIN {X 0,Y 341.295,Z 140.783,A -85,B 0,C 180,E1 -14040,E2 -14040} C_VEL
LIN {X 0,Y 341.167,Z 140.798,A -85,B 0,C 180,E1 -14042.361,E2 -14042.361} C_VEL
LIN {X 0,Y 341.076,Z 140.809,A -85,B 0,C 180,E1 -14047.102,E2 -14047.102} C_VEL
LIN {X 0,Y 340.869,Z 140.831,A -85,B 0,C 180,E1 -14050.694,E2 -14050.694} C_VEL
LIN {X 0,Y 340.861,Z 140.835,A -85,B 0,C 180,E1 -14054.325,E2 -14054.325} C_VEL
LIN {X 0,Y 340.835,Z 140.837,A -85,B 0,C 180,E1 -14058.466,E2 -14058.466} C_VEL
LIN {X 0,Y 340.752,Z 140.849,A -85,B 0,C 180,E1 -14061.857,E2 -14061.857} C_VEL
LIN {X 0,Y 340.771,Z 140.846,A -85,B 0,C 180,E1 -14065.664,E2 -14065.664} C_VEL
LIN {X 0,Y 340.739,Z 140.849,A -85,B 0,C 180,E1 -14068.32,E2 -14068.32} C_VEL
LIN {X 0,Y 340.702,Z 140.859,A -85,B 0,C 180,E1 -14071.044,E2 -14071.044} C_VEL
LIN {X 0,Y 340.716,Z 140.853,A -85,B 0,C 180,E1 -14075.279,E2 -14075.279} C_VEL
LIN {X 0,Y 340.708,Z 140.859,A -85,B 0,C 180,E1 -14078.386,E2 -14078.386} C_VEL
LIN {X 0,Y 340.697,Z 140.856,A -85,B 0,C 180,E1 -14082.046,E2 -14082.046} C_VEL
LIN {X 0,Y 340.65,Z 140.866,A -85,B 0,C 180,E1 -14086.227,E2 -14086.227} C_VEL
LIN {X 0,Y 340.687,Z 140.86,A -85,B 0,C 180,E1 -14089.753,E2 -14089.753} C_VEL
LIN {X 0,Y 340.703,Z 140.855,A -85,B 0,C 180,E1 -14093.259,E2 -14093.259} C_VEL
LIN {X 0,Y 340.692,Z 140.857,A -85,B 0,C 180,E1 -14096.154,E2 -14096.154} C_VEL
LIN {X 0,Y 340.773,Z 140.844,A -85,B 0,C 180,E1 -14100.333,E2 -14100.333} C_VEL
LIN {X 0,Y 340.873,Z 141.051,A -85,B 0,C 180,E1 -14103.522,E2 -14103.522} C_VEL
LIN {X 0,Y 342.66,Z 150.996,A -85,B 0,C 180,E1 -14106.746,E2 -14106.746} C_VEL
LIN {X 0,Y 342.895,Z 154.458,A -85,B 0,C 180,E1 -14107.812,E2 -14107.812} C_VEL
LIN {X 0,Y 341.674,Z 167.049,A -85,B 0,C 180,E1 -14111.472,E2 -14111.472} C_VEL
LIN {X 0,Y 342.089,Z 169.847,A -85,B 0,C 180,E1 -14111.63,E2 -14111.63} C_VEL
LIN {X 0,Y 345.7,Z 193.314,A -85,B 0,C 180,E1 -14112.329,E2 -14112.329} C_VEL
LIN {X 0,Y 346.152,Z 198.545,A -85,B 0,C 180,E1 -14112.464,E2 -14112.464} C_VEL
LIN {X 0,Y 345.529,Z 244.012,A -85,B 0,C 180,E1 -14113.434,E2 -14113.434} C_VEL
LIN {X 0,Y 345.064,Z 253.454,A -85,B 0,C 180,E1 -14113.775,E2 -14113.775} C_VEL
LIN {X 0,Y 344.52,Z 263.465,A -85,B 0,C 180,E1 -14114.319,E2 -14114.319} C_VEL
LIN {X 0,Y 343.626,Z 274.837,A -85,B 0,C 180,E1 -14115.188,E2 -14115.188} C_VEL
LIN {X 0,Y 342.9,Z 283.412,A -85,B 0,C 180,E1 -14116.065,E2 -14116.065} C_VEL
LIN {X 0,Y 342.051,Z 291.479,A -85,B 0,C 180,E1 -14117.089,E2 -14117.089} C_VEL
LIN {X 0,Y 341.395,Z 298.144,A -85,B 0,C 180,E1 -14118.12,E2 -14118.12} C_VEL
LIN {X 0,Y 340.745,Z 304.473,A -85,B 0,C 180,E1 -14119.303,E2 -14119.303} C_VEL
LIN {X 0,Y 340.215,Z 309.731,A -85,B 0,C 180,E1 -14120.488,E2 -14120.488} C_VEL
LIN {X 0,Y 339.796,Z 314.116,A -85,B 0,C 180,E1 -14121.676,E2 -14121.676} C_VEL
LIN {X 0,Y 339.36,Z 319.44,A -85,B 0,C 180,E1 -14123.52,E2 -14123.52} C_VEL
LIN {X 0,Y 339.158,Z 323.086,A -85,B 0,C 180,E1 -14125.246,E2 -14125.246} C_VEL
LIN {X 0,Y 339.082,Z 324.831,A -85,B 0,C 180,E1 -14126.435,E2 -14126.435} C_VEL
LIN {X 0,Y 338.981,Z 326.079,A -85,B 0,C 180,E1 -14127.624,E2 -14127.624} C_VEL
LIN {X 0,Y 338.961,Z 326.856,A -85,B 0,C 180,E1 -14128.812,E2 -14128.812} C_VEL
LIN {X 0,Y 338.994,Z 327.15,A -85,B 0,C 180,E1 -14130,E2 -14130} C_VEL
LIN {X 0,Y 338.961,Z 326.851,A -85,B 0,C 180,E1 -14131.188,E2 -14131.188} C_VEL
LIN {X 0,Y 338.981,Z 326.065,A -85,B 0,C 180,E1 -14132.377,E2 -14132.377} C_VEL
LIN {X 0,Y 339.082,Z 324.807,A -85,B 0,C 180,E1 -14133.565,E2 -14133.565} C_VEL
LIN {X 0,Y 339.158,Z 323.051,A -85,B 0,C 180,E1 -14134.755,E2 -14134.755} C_VEL
LIN {X 0,Y 339.364,Z 319.395,A -85,B 0,C 180,E1 -14136.481,E2 -14136.481} C_VEL
LIN {X 0,Y 339.72,Z 314.055,A -85,B 0,C 180,E1 -14138.327,E2 -14138.327} C_VEL
LIN {X 0,Y 340.482,Z 307.221,A -85,B 0,C 180,E1 -14140.105,E2 -14140.105} C_VEL
LIN {X 0,Y 341.206,Z 299.751,A -85,B 0,C 180,E1 -14141.586,E2 -14141.586} C_VEL
LIN {X 0,Y 341.959,Z 292.384,A -85,B 0,C 180,E1 -14142.764,E2 -14142.764} C_VEL
LIN {X 0,Y 342.733,Z 284.495,A -85,B 0,C 180,E1 -14143.791,E2 -14143.791} C_VEL
LIN {X 0,Y 343.486,Z 276.156,A -85,B 0,C 180,E1 -14144.667,E2 -14144.667} C_VEL
LIN {X 0,Y 344.327,Z 265.499,A -85,B 0,C 180,E1 -14145.539,E2 -14145.539} C_VEL
LIN {X 0,Y 345.002,Z 253.879,A -85,B 0,C 180,E1 -14146.19,E2 -14146.19} C_VEL
LIN {X 0,Y 345.495,Z 244.124,A -85,B 0,C 180,E1 -14146.546,E2 -14146.546} C_VEL
LIN {X 0,Y 346.017,Z 195.731,A -85,B 0,C 180,E1 -14147.584,E2 -14147.584} C_VEL
LIN {X 0,Y 342.046,Z 169.663,A -85,B 0,C 180,E1 -14148.357,E2 -14148.357} C_VEL
LIN {X 0,Y 341.688,Z 167.188,A -85,B 0,C 180,E1 -14148.49,E2 -14148.49} C_VEL
LIN {X 0,Y 342.872,Z 154.417,A -85,B 0,C 180,E1 -14152.182,E2 -14152.182} C_VEL
LIN {X 0,Y 342.468,Z 149.873,A -85,B 0,C 180,E1 -14153.589,E2 -14153.589} C_VEL
LIN {X 0,Y 340.83,Z 140.879,A -85,B 0,C 180,E1 -14156.565,E2 -14156.565} C_VEL
LIN {X 0,Y 340.764,Z 140.848,A -85,B 0,C 180,E1 -14159.978,E2 -14159.978} C_VEL
LIN {X 0,Y 340.692,Z 140.856,A -85,B 0,C 180,E1 -14163.847,E2 -14163.847} C_VEL
LIN {X 0,Y 340.705,Z 140.854,A -85,B 0,C 180,E1 -14166.742,E2 -14166.742} C_VEL
LIN {X 0,Y 340.689,Z 140.86,A -85,B 0,C 180,E1 -14170.247,E2 -14170.247} C_VEL
LIN {X 0,Y 340.652,Z 140.865,A -85,B 0,C 180,E1 -14173.773,E2 -14173.773} C_VEL
LIN {X 0,Y 340.699,Z 140.856,A -85,B 0,C 180,E1 -14177.955,E2 -14177.955} C_VEL
LIN {X 0,Y 340.733,Z 140.855,A -85,B 0,C 180,E1 -14181.773,E2 -14181.773} C_VEL
LIN {X 0,Y 340.724,Z 140.855,A -85,B 0,C 180,E1 -14185.596,E2 -14185.596} C_VEL
LIN {X 0,Y 340.705,Z 140.858,A -85,B 0,C 180,E1 -14188.956,E2 -14188.956} C_VEL
LIN {X 0,Y 340.78,Z 140.844,A -85,B 0,C 180,E1 -14192.474,E2 -14192.474} C_VEL
LIN {X 0,Y 340.757,Z 140.849,A -85,B 0,C 180,E1 -14195.639,E2 -14195.639} C_VEL
LIN {X 0,Y 340.754,Z 140.847,A -85,B 0,C 180,E1 -14199.475,E2 -14199.475} C_VEL
LIN {X 0,Y 340.859,Z 140.834,A -85,B 0,C 180,E1 -14201.984,E2 -14201.984} C_VEL
LIN {X 0,Y 340.871,Z 140.834,A -85,B 0,C 180,E1 -14205.705,E2 -14205.705} C_VEL
LIN {X 0,Y 340.873,Z 140.831,A -85,B 0,C 180,E1 -14209.306,E2 -14209.306} C_VEL
LIN {X 0,Y 341.06,Z 140.812,A -85,B 0,C 180,E1 -14212.898,E2 -14212.898} C_VEL
LIN {X 0,Y 341.169,Z 140.797,A -85,B 0,C 180,E1 -14217.639,E2 -14217.639} C_VEL
LIN {X 0,Y 341.277,Z 140.785,A -85,B 0,C 180,E1 -14220,E2 -14220} C_VEL
LIN {X 0,Y 341.169,Z 140.799,A -85,B 0,C 180,E1 -14222.361,E2 -14222.361} C_VEL
LIN {X 0,Y 341.078,Z 140.808,A -85,B 0,C 180,E1 -14227.102,E2 -14227.102} C_VEL
LIN {X 0,Y 340.877,Z 140.832,A -85,B 0,C 180,E1 -14230.694,E2 -14230.694} C_VEL
LIN {X 0,Y 340.865,Z 140.835,A -85,B 0,C 180,E1 -14234.325,E2 -14234.325} C_VEL
LIN {X 0,Y 340.839,Z 140.835,A -85,B 0,C 180,E1 -14238.466,E2 -14238.466} C_VEL
LIN {X 0,Y 340.755,Z 140.849,A -85,B 0,C 180,E1 -14241.857,E2 -14241.857} C_VEL
LIN {X 0,Y 340.774,Z 140.845,A -85,B 0,C 180,E1 -14245.664,E2 -14245.664} C_VEL
LIN {X 0,Y 340.742,Z 140.85,A -85,B 0,C 180,E1 -14248.32,E2 -14248.32} C_VEL
LIN {X 0,Y 340.705,Z 140.859,A -85,B 0,C 180,E1 -14251.044,E2 -14251.044} C_VEL
LIN {X 0,Y 340.72,Z 140.854,A -85,B 0,C 180,E1 -14255.279,E2 -14255.279} C_VEL
LIN {X 0,Y 340.711,Z 140.858,A -85,B 0,C 180,E1 -14258.386,E2 -14258.386} C_VEL
LIN {X 0,Y 340.7,Z 140.857,A -85,B 0,C 180,E1 -14262.045,E2 -14262.045} C_VEL
LIN {X 0,Y 340.653,Z 140.864,A -85,B 0,C 180,E1 -14266.227,E2 -14266.227} C_VEL
LIN {X 0,Y 340.69,Z 140.857,A -85,B 0,C 180,E1 -14269.753,E2 -14269.753} C_VEL
LIN {X 0,Y 340.707,Z 140.854,A -85,B 0,C 180,E1 -14273.258,E2 -14273.258} C_VEL
LIN {X 0,Y 340.696,Z 140.86,A -85,B 0,C 180,E1 -14276.154,E2 -14276.154} C_VEL
LIN {X 0,Y 340.776,Z 140.847,A -85,B 0,C 180,E1 -14280.332,E2 -14280.332} C_VEL
LIN {X 0,Y 340.807,Z 140.843,A -85,B 0,C 180,E1 -14283.02,E2 -14283.02} C_VEL
LIN {X 0,Y 340.79,Z 140.996,A -85,B 0,C 180,E1 -14286.771,E2 -14286.771} C_VEL
LIN {X 0,Y 341.919,Z 147.225,A -85,B 0,C 180,E1 -14288.918,E2 -14288.918} C_VEL
LIN {X 0,Y 342.086,Z 153.082,A -85,B 0,C 180,E1 -14290.809,E2 -14290.809} C_VEL
LIN {X 0,Y 341.998,Z 155.629,A -85,B 0,C 180,E1 -14291.562,E2 -14291.562} C_VEL
LIN {X 0,Y 342.236,Z 157.482,A -85,B 0,C 180,E1 -14291.689,E2 -14291.689} C_VEL
LIN {X 0,Y 346.351,Z 180.22,A -85,B 0,C 180,E1 -14292.402,E2 -14292.402} C_VEL
LIN {X 0,Y 345.558,Z 231.897,A -85,B 0,C 180,E1 -14293.495,E2 -14293.495} C_VEL
LIN {X 0,Y 345.211,Z 241.731,A -85,B 0,C 180,E1 -14293.858,E2 -14293.858} C_VEL
LIN {X 0,Y 344.727,Z 252.844,A -85,B 0,C 180,E1 -14294.479,E2 -14294.479} C_VEL
LIN {X 0,Y 343.934,Z 263.678,A -85,B 0,C 180,E1 -14295.352,E2 -14295.352} C_VEL
LIN {X 0,Y 343.138,Z 272.077,A -85,B 0,C 180,E1 -14296.225,E2 -14296.225} C_VEL
LIN {X 0,Y 342.48,Z 280.002,A -85,B 0,C 180,E1 -14297.255,E2 -14297.255} C_VEL
LIN {X 0,Y 341.875,Z 285.695,A -85,B 0,C 180,E1 -14298.137,E2 -14298.137} C_VEL
LIN {X 0,Y 341.187,Z 292.05,A -85,B 0,C 180,E1 -14299.316,E2 -14299.316} C_VEL
LIN {X 0,Y 340.572,Z 297.332,A -85,B 0,C 180,E1 -14300.497,E2 -14300.497} C_VEL
LIN {X 0,Y 340.183,Z 301.74,A -85,B 0,C 180,E1 -14301.685,E2 -14301.685} C_VEL
LIN {X 0,Y 339.805,Z 305.994,A -85,B 0,C 180,E1 -14303.102,E2 -14303.102} C_VEL
LIN {X 0,Y 339.497,Z 309.583,A -85,B 0,C 180,E1 -14304.655,E2 -14304.655} C_VEL
LIN {X 0,Y 339.185,Z 312.498,A -85,B 0,C 180,E1 -14306.436,E2 -14306.436} C_VEL
LIN {X 0,Y 339.047,Z 313.772,A -85,B 0,C 180,E1 -14307.624,E2 -14307.624} C_VEL
LIN {X 0,Y 338.991,Z 314.576,A -85,B 0,C 180,E1 -14308.812,E2 -14308.812} C_VEL
LIN {X 0,Y 338.998,Z 314.882,A -85,B 0,C 180,E1 -14310,E2 -14310} C_VEL
LIN {X 0,Y 338.991,Z 314.605,A -85,B 0,C 180,E1 -14311.188,E2 -14311.188} C_VEL
LIN {X 0,Y 339.046,Z 313.86,A -85,B 0,C 180,E1 -14312.376,E2 -14312.376} C_VEL
LIN {X 0,Y 339.181,Z 312.645,A -85,B 0,C 180,E1 -14313.564,E2 -14313.564} C_VEL
LIN {X 0,Y 339.48,Z 309.792,A -85,B 0,C 180,E1 -14315.345,E2 -14315.345} C_VEL
LIN {X 0,Y 339.719,Z 306.578,A -85,B 0,C 180,E1 -14316.778,E2 -14316.778} C_VEL
LIN {X 0,Y 340.158,Z 302.087,A -85,B 0,C 180,E1 -14318.315,E2 -14318.315} C_VEL
LIN {X 0,Y 340.689,Z 296.59,A -85,B 0,C 180,E1 -14319.798,E2 -14319.798} C_VEL
LIN {X 0,Y 341.48,Z 289.682,A -85,B 0,C 180,E1 -14321.275,E2 -14321.275} C_VEL
LIN {X 0,Y 342.283,Z 281.749,A -85,B 0,C 180,E1 -14322.601,E2 -14322.601} C_VEL
LIN {X 0,Y 343.053,Z 274.183,A -85,B 0,C 180,E1 -14323.626,E2 -14323.626} C_VEL
LIN {X 0,Y 343.801,Z 266.252,A -85,B 0,C 180,E1 -14324.502,E2 -14324.502} C_VEL
LIN {X 0,Y 344.382,Z 258.061,A -85,B 0,C 180,E1 -14325.233,E2 -14325.233} C_VEL
LIN {X 0,Y 344.947,Z 249.759,A -85,B 0,C 180,E1 -14325.813,E2 -14325.813} C_VEL
LIN {X 0,Y 345.345,Z 240.786,A -85,B 0,C 180,E1 -14326.287,E2 -14326.287} C_VEL
LIN {X 0,Y 345.659,Z 231.542,A -85,B 0,C 180,E1 -14326.619,E2 -14326.619} C_VEL
LIN {X 0,Y 346.289,Z 179.58,A -85,B 0,C 180,E1 -14327.723,E2 -14327.723} C_VEL
LIN {X 0,Y 341.997,Z 156.053,A -85,B 0,C 180,E1 -14328.495,E2 -14328.495} C_VEL
LIN {X 0,Y 341.993,Z 154.919,A -85,B 0,C 180,E1 -14328.724,E2 -14328.724} C_VEL
LIN {X 0,Y 342.14,Z 149.522,A -85,B 0,C 180,E1 -14330.438,E2 -14330.438} C_VEL
LIN {X 0,Y 341.282,Z 143.491,A -85,B 0,C 180,E1 -14332.456,E2 -14332.456} C_VEL
LIN {X 0,Y 340.77,Z 140.953,A -85,B 0,C 180,E1 -14333.391,E2 -14333.391} C_VEL
LIN {X 0,Y 340.805,Z 140.843,A -85,B 0,C 180,E1 -14336.98,E2 -14336.98} C_VEL
LIN {X 0,Y 340.78,Z 140.845,A -85,B 0,C 180,E1 -14337.479,E2 -14337.479} C_VEL
LIN {X 0,Y 340.099,Z 140.935,A -85,B 0,C 180,E1 -14338.465,E2 -14338.465} C_VEL
LIN {X 0,Y 337.224,Z 141.295,A -85,B 0,C 180,E1 -14340.067,E2 -14340.067} C_VEL
LIN {X 0,Y 334.787,Z 141.598,A -85,B 0,C 180,E1 -14341.365,E2 -14341.365} C_VEL
LIN {X 0,Y 333.732,Z 141.727,A -85,B 0,C 180,E1 -14342.37,E2 -14342.37} C_VEL
LIN {X 0,Y 333.641,Z 141.736,A -85,B 0,C 180,E1 -14342.71,E2 -14342.71} C_VEL
LIN {X 0,Y 333.676,Z 141.732,A -85,B 0,C 180,E1 -14346.138,E2 -14346.138} C_VEL
LIN {X 0,Y 333.647,Z 141.735,A -85,B 0,C 180,E1 -14349.192,E2 -14349.192} C_VEL
LIN {X 0,Y 333.632,Z 141.728,A -85,B 0,C 180,E1 -14352.5,E2 -14352.5} C_VEL
LIN {X 0,Y 333.596,Z 141.744,A -85,B 0,C 180,E1 -14355.955,E2 -14355.955} C_VEL
LIN {X 0,Y 333.646,Z 141.738,A -85,B 0,C 180,E1 -14359.315,E2 -14359.315} C_VEL
LIN {X 0,Y 333.664,Z 141.736,A -85,B 0,C 180,E1 -14363.167,E2 -14363.167} C_VEL
LIN {X 0,Y 333.673,Z 141.733,A -85,B 0,C 180,E1 -14365.341,E2 -14365.341} C_VEL
LIN {X 0,Y 333.701,Z 141.728,A -85,B 0,C 180,E1 -14369.71,E2 -14369.71} C_VEL
LIN {X 0,Y 333.741,Z 141.722,A -85,B 0,C 180,E1 -14372.401,E2 -14372.401} C_VEL
LIN {X 0,Y 333.726,Z 141.728,A -85,B 0,C 180,E1 -14375.09,E2 -14375.09} C_VEL
LIN {X 0,Y 333.684,Z 141.732,A -85,B 0,C 180,E1 -14379.019,E2 -14379.019} C_VEL
LIN {X 0,Y 333.792,Z 141.712,A -85,B 0,C 180,E1 -14381.589,E2 -14381.589} C_VEL
LIN {X 0,Y 333.807,Z 141.714,A -85,B 0,C 180,E1 -14385.576,E2 -14385.576} C_VEL
LIN {X 0,Y 333.836,Z 141.709,A -85,B 0,C 180,E1 -14389.078,E2 -14389.078} C_VEL
LIN {X 0,Y 334.024,Z 141.687,A -85,B 0,C 180,E1 -14392.747,E2 -14392.747} C_VEL
LIN {X 0,Y 333.809,Z 141.714,A -85,B 0,C 180,E1 -14395.169,E2 -14395.169} C_VEL
LIN {X 0,Y 334.105,Z 141.678,A -85,B 0,C 180,E1 -14397.589,E2 -14397.589} C_VEL
LIN {X 0,Y 334.246,Z 141.66,A -85,B 0,C 180,E1 -14400,E2 -14400} C_VEL
LIN {X 0,Y 334.104,Z 141.677,A -85,B 0,C 180,E1 -14402.411,E2 -14402.411} C_VEL
LIN {X 0,Y 334.022,Z 141.69,A -85,B 0,C 180,E1 -14406.039,E2 -14406.039} C_VEL
LIN {X 0,Y 333.983,Z 141.69,A -85,B 0,C 180,E1 -14408.501,E2 -14408.501} C_VEL
LIN {X 0,Y 333.789,Z 141.716,A -85,B 0,C 180,E1 -14412.155,E2 -14412.155} C_VEL
LIN {X 0,Y 333.776,Z 141.719,A -85,B 0,C 180,E1 -14415.886,E2 -14415.886} C_VEL
LIN {X 0,Y 333.794,Z 141.715,A -85,B 0,C 180,E1 -14418.655,E2 -14418.655} C_VEL
LIN {X 0,Y 333.69,Z 141.728,A -85,B 0,C 180,E1 -14422.278,E2 -14422.278} C_VEL
LIN {X 0,Y 333.734,Z 141.723,A -85,B 0,C 180,E1 -14426.246,E2 -14426.246} C_VEL
LIN {X 0,Y 333.709,Z 141.73,A -85,B 0,C 180,E1 -14428.972,E2 -14428.972} C_VEL
LIN {X 0,Y 333.641,Z 141.739,A -85,B 0,C 180,E1 -14432.587,E2 -14432.587} C_VEL
LIN {X 0,Y 333.674,Z 141.731,A -85,B 0,C 180,E1 -14436.139,E2 -14436.139} C_VEL
LIN {X 0,Y 333.645,Z 141.734,A -85,B 0,C 180,E1 -14439.192,E2 -14439.192} C_VEL
LIN {X 0,Y 333.63,Z 141.731,A -85,B 0,C 180,E1 -14442.5,E2 -14442.5} C_VEL
LIN {X 0,Y 333.594,Z 141.741,A -85,B 0,C 180,E1 -14445.955,E2 -14445.955} C_VEL
LIN {X 0,Y 333.645,Z 141.734,A -85,B 0,C 180,E1 -14449.316,E2 -14449.316} C_VEL
LIN {X 0,Y 333.664,Z 141.731,A -85,B 0,C 180,E1 -14453.168,E2 -14453.168} C_VEL
LIN {X 0,Y 333.637,Z 141.733,A -85,B 0,C 180,E1 -14456.792,E2 -14456.792} C_VEL
LIN {X 0,Y 333.701,Z 141.73,A -85,B 0,C 180,E1 -14459.711,E2 -14459.711} C_VEL
LIN {X 0,Y 333.815,Z 141.799,A -85,B 0,C 180,E1 -14463.171,E2 -14463.171} C_VEL
LIN {X 0,Y 335.646,Z 151.916,A -85,B 0,C 180,E1 -14466.557,E2 -14466.557} C_VEL
LIN {X 0,Y 335.842,Z 156.114,A -85,B 0,C 180,E1 -14467.872,E2 -14467.872} C_VEL
LIN {X 0,Y 334.744,Z 167.009,A -85,B 0,C 180,E1 -14471.088,E2 -14471.088} C_VEL
LIN {X 0,Y 335.403,Z 171.105,A -85,B 0,C 180,E1 -14471.281,E2 -14471.281} C_VEL
LIN {X 0,Y 338.934,Z 193.974,A -85,B 0,C 180,E1 -14471.981,E2 -14471.981} C_VEL
LIN {X 0,Y 339.393,Z 198.675,A -85,B 0,C 180,E1 -14472.109,E2 -14472.109} C_VEL
LIN {X 0,Y 338.733,Z 243.244,A -85,B 0,C 180,E1 -14473.072,E2 -14473.072} C_VEL
LIN {X 0,Y 338.318,Z 252.504,A -85,B 0,C 180,E1 -14473.404,E2 -14473.404} C_VEL
LIN {X 0,Y 337.758,Z 262.133,A -85,B 0,C 180,E1 -14473.919,E2 -14473.919} C_VEL
LIN {X 0,Y 337.069,Z 271.273,A -85,B 0,C 180,E1 -14474.583,E2 -14474.583} C_VEL
LIN {X 0,Y 336.147,Z 282.055,A -85,B 0,C 180,E1 -14475.625,E2 -14475.625} C_VEL
LIN {X 0,Y 335.236,Z 290.331,A -85,B 0,C 180,E1 -14476.667,E2 -14476.667} C_VEL
LIN {X 0,Y 334.43,Z 298.018,A -85,B 0,C 180,E1 -14477.869,E2 -14477.869} C_VEL
LIN {X 0,Y 333.748,Z 304.346,A -85,B 0,C 180,E1 -14479.076,E2 -14479.076} C_VEL
LIN {X 0,Y 333.186,Z 309.604,A -85,B 0,C 180,E1 -14480.285,E2 -14480.285} C_VEL
LIN {X 0,Y 332.756,Z 313.989,A -85,B 0,C 180,E1 -14481.498,E2 -14481.498} C_VEL
LIN {X 0,Y 332.316,Z 319.161,A -85,B 0,C 180,E1 -14483.321,E2 -14483.321} C_VEL
LIN {X 0,Y 332.063,Z 322.958,A -85,B 0,C 180,E1 -14485.144,E2 -14485.144} C_VEL
LIN {X 0,Y 332.011,Z 324.704,A -85,B 0,C 180,E1 -14486.359,E2 -14486.359} C_VEL
LIN {X 0,Y 331.9,Z 325.952,A -85,B 0,C 180,E1 -14487.573,E2 -14487.573} C_VEL
LIN {X 0,Y 331.869,Z 326.728,A -85,B 0,C 180,E1 -14488.787,E2 -14488.787} C_VEL
LIN {X 0,Y 331.899,Z 327.022,A -85,B 0,C 180,E1 -14490,E2 -14490} C_VEL
LIN {X 0,Y 331.869,Z 326.723,A -85,B 0,C 180,E1 -14491.214,E2 -14491.214} C_VEL
LIN {X 0,Y 331.901,Z 325.936,A -85,B 0,C 180,E1 -14492.427,E2 -14492.427} C_VEL
LIN {X 0,Y 332.011,Z 324.678,A -85,B 0,C 180,E1 -14493.641,E2 -14493.641} C_VEL
LIN {X 0,Y 332.098,Z 321.608,A -85,B 0,C 180,E1 -14495.548,E2 -14495.548} C_VEL
LIN {X 0,Y 332.419,Z 317.591,A -85,B 0,C 180,E1 -14497.288,E2 -14497.288} C_VEL
LIN {X 0,Y 332.933,Z 311.876,A -85,B 0,C 180,E1 -14499.11,E2 -14499.11} C_VEL
LIN {X 0,Y 333.585,Z 305.674,A -85,B 0,C 180,E1 -14500.623,E2 -14500.623} C_VEL
LIN {X 0,Y 334.247,Z 299.62,A -85,B 0,C 180,E1 -14501.83,E2 -14501.83} C_VEL
LIN {X 0,Y 335.043,Z 292.253,A -85,B 0,C 180,E1 -14503.032,E2 -14503.032} C_VEL
LIN {X 0,Y 335.85,Z 284.363,A -85,B 0,C 180,E1 -14504.08,E2 -14504.08} C_VEL
LIN {X 0,Y 336.627,Z 276.024,A -85,B 0,C 180,E1 -14504.973,E2 -14504.973} C_VEL
LIN {X 0,Y 337.499,Z 265.365,A -85,B 0,C 180,E1 -14505.862,E2 -14505.862} C_VEL
LIN {X 0,Y 338.211,Z 253.742,A -85,B 0,C 180,E1 -14506.525,E2 -14506.525} C_VEL
LIN {X 0,Y 338.715,Z 243.981,A -85,B 0,C 180,E1 -14506.887,E2 -14506.887} C_VEL
LIN {X 0,Y 339.266,Z 196.495,A -85,B 0,C 180,E1 -14507.926,E2 -14507.926} C_VEL
LIN {X 0,Y 335.225,Z 170.149,A -85,B 0,C 180,E1 -14508.73,E2 -14508.73} C_VEL
LIN {X 0,Y 334.74,Z 167.142,A -85,B 0,C 180,E1 -14508.873,E2 -14508.873} C_VEL
LIN {X 0,Y 335.53,Z 159.179,A -85,B 0,C 180,E1 -14511.181,E2 -14511.181} C_VEL
LIN {X 0,Y 335.83,Z 153.365,A -85,B 0,C 180,E1 -14512.957,E2 -14512.957} C_VEL
LIN {X 0,Y 334.109,Z 143.413,A -85,B 0,C 180,E1 -14516.215,E2 -14516.215} C_VEL
LIN {X 0,Y 333.78,Z 141.74,A -85,B 0,C 180,E1 -14516.875,E2 -14516.875} C_VEL
LIN {X 0,Y 333.698,Z 141.731,A -85,B 0,C 180,E1 -14520.362,E2 -14520.362} C_VEL
LIN {X 0,Y 333.686,Z 141.731,A -85,B 0,C 180,E1 -14524.774,E2 -14524.774} C_VEL
LIN {X 0,Y 333.652,Z 141.734,A -85,B 0,C 180,E1 -14527.651,E2 -14527.651} C_VEL
LIN {X 0,Y 333.647,Z 141.734,A -85,B 0,C 180,E1 -14530.768,E2 -14530.768} C_VEL
LIN {X 0,Y 333.593,Z 141.739,A -85,B 0,C 180,E1 -14534.251,E2 -14534.251} C_VEL
LIN {X 0,Y 333.642,Z 141.731,A -85,B 0,C 180,E1 -14537.619,E2 -14537.619} C_VEL
LIN {X 0,Y 333.653,Z 141.736,A -85,B 0,C 180,E1 -14541.202,E2 -14541.202} C_VEL
LIN {X 0,Y 333.677,Z 141.731,A -85,B 0,C 180,E1 -14543.861,E2 -14543.861} C_VEL
LIN {X 0,Y 333.644,Z 141.739,A -85,B 0,C 180,E1 -14547.413,E2 -14547.413} C_VEL
LIN {X 0,Y 333.712,Z 141.73,A -85,B 0,C 180,E1 -14551.028,E2 -14551.028} C_VEL
LIN {X 0,Y 333.737,Z 141.722,A -85,B 0,C 180,E1 -14553.754,E2 -14553.754} C_VEL
LIN {X 0,Y 333.721,Z 141.724,A -85,B 0,C 180,E1 -14557.914,E2 -14557.914} C_VEL
LIN {X 0,Y 333.795,Z 141.714,A -85,B 0,C 180,E1 -14561.59,E2 -14561.59} C_VEL
LIN {X 0,Y 333.81,Z 141.714,A -85,B 0,C 180,E1 -14565.577,E2 -14565.577} C_VEL
LIN {X 0,Y 333.835,Z 141.707,A -85,B 0,C 180,E1 -14569.078,E2 -14569.078} C_VEL
LIN {X 0,Y 334.007,Z 141.691,A -85,B 0,C 180,E1 -14572.747,E2 -14572.747} C_VEL
LIN {X 0,Y 333.809,Z 141.714,A -85,B 0,C 180,E1 -14575.169,E2 -14575.169} C_VEL
LIN {X 0,Y 334.106,Z 141.676,A -85,B 0,C 180,E1 -14577.589,E2 -14577.589} C_VEL
LIN {X 0,Y 334.229,Z 141.662,A -85,B 0,C 180,E1 -14580,E2 -14580} C_VEL
LIN {X 0,Y 334.106,Z 141.678,A -85,B 0,C 180,E1 -14582.411,E2 -14582.411} C_VEL
LIN {X 0,Y 334.027,Z 141.686,A -85,B 0,C 180,E1 -14587.253,E2 -14587.253} C_VEL
LIN {X 0,Y 333.84,Z 141.708,A -85,B 0,C 180,E1 -14590.922,E2 -14590.922} C_VEL
LIN {X 0,Y 333.81,Z 141.714,A -85,B 0,C 180,E1 -14594.634,E2 -14594.634} C_VEL
LIN {X 0,Y 333.798,Z 141.712,A -85,B 0,C 180,E1 -14598.655,E2 -14598.655} C_VEL
LIN {X 0,Y 333.694,Z 141.728,A -85,B 0,C 180,E1 -14602.278,E2 -14602.278} C_VEL
LIN {X 0,Y 333.737,Z 141.72,A -85,B 0,C 180,E1 -14606.246,E2 -14606.246} C_VEL
LIN {X 0,Y 333.712,Z 141.73,A -85,B 0,C 180,E1 -14608.972,E2 -14608.972} C_VEL
LIN {X 0,Y 333.645,Z 141.737,A -85,B 0,C 180,E1 -14612.587,E2 -14612.587} C_VEL
LIN {X 0,Y 333.678,Z 141.731,A -85,B 0,C 180,E1 -14616.139,E2 -14616.139} C_VEL
LIN {X 0,Y 333.648,Z 141.733,A -85,B 0,C 180,E1 -14619.192,E2 -14619.192} C_VEL
LIN {X 0,Y 333.634,Z 141.742,A -85,B 0,C 180,E1 -14622.5,E2 -14622.5} C_VEL
LIN {X 0,Y 333.598,Z 141.741,A -85,B 0,C 180,E1 -14625.955,E2 -14625.955} C_VEL
LIN {X 0,Y 333.649,Z 141.731,A -85,B 0,C 180,E1 -14629.315,E2 -14629.315} C_VEL
LIN {X 0,Y 333.667,Z 141.731,A -85,B 0,C 180,E1 -14633.168,E2 -14633.168} C_VEL
LIN {X 0,Y 333.641,Z 141.735,A -85,B 0,C 180,E1 -14636.792,E2 -14636.792} C_VEL
LIN {X 0,Y 333.704,Z 141.73,A -85,B 0,C 180,E1 -14639.71,E2 -14639.71} C_VEL
LIN {X 0,Y 333.745,Z 141.722,A -85,B 0,C 180,E1 -14642.401,E2 -14642.401} C_VEL
LIN {X 0,Y 333.757,Z 141.827,A -85,B 0,C 180,E1 -14646.457,E2 -14646.457} C_VEL
LIN {X 0,Y 335.04,Z 149.299,A -85,B 0,C 180,E1 -14649.108,E2 -14649.108} C_VEL
LIN {X 0,Y 335.08,Z 155.178,A -85,B 0,C 180,E1 -14651.028,E2 -14651.028} C_VEL
LIN {X 0,Y 335.147,Z 156.521,A -85,B 0,C 180,E1 -14651.25,E2 -14651.25} C_VEL
LIN {X 0,Y 339.511,Z 180.542,A -85,B 0,C 180,E1 -14652.039,E2 -14652.039} C_VEL
LIN {X 0,Y 338.766,Z 232.043,A -85,B 0,C 180,E1 -14653.154,E2 -14653.154} C_VEL
LIN {X 0,Y 338.419,Z 241.87,A -85,B 0,C 180,E1 -14653.524,E2 -14653.524} C_VEL
LIN {X 0,Y 337.9,Z 252.98,A -85,B 0,C 180,E1 -14654.158,E2 -14654.158} C_VEL
LIN {X 0,Y 337.074,Z 263.812,A -85,B 0,C 180,E1 -14655.047,E2 -14655.047} C_VEL
LIN {X 0,Y 336.27,Z 272.209,A -85,B 0,C 180,E1 -14655.938,E2 -14655.938} C_VEL
LIN {X 0,Y 335.581,Z 280.134,A -85,B 0,C 180,E1 -14656.989,E2 -14656.989} C_VEL
LIN {X 0,Y 334.924,Z 285.826,A -85,B 0,C 180,E1 -14657.887,E2 -14657.887} C_VEL
LIN {X 0,Y 334.229,Z 292.18,A -85,B 0,C 180,E1 -14659.091,E2 -14659.091} C_VEL
LIN {X 0,Y 333.446,Z 298.632,A -85,B 0,C 180,E1 -14660.599,E2 -14660.599} C_VEL
LIN {X 0,Y 332.979,Z 303.777,A -85,B 0,C 180,E1 -14662.114,E2 -14662.114} C_VEL
LIN {X 0,Y 332.509,Z 308.538,A -85,B 0,C 180,E1 -14663.933,E2 -14663.933} C_VEL
LIN {X 0,Y 332.323,Z 310.86,A -85,B 0,C 180,E1 -14665.147,E2 -14665.147} C_VEL
LIN {X 0,Y 332.117,Z 312.627,A -85,B 0,C 180,E1 -14666.36,E2 -14666.36} C_VEL
LIN {X 0,Y 331.965,Z 313.901,A -85,B 0,C 180,E1 -14667.573,E2 -14667.573} C_VEL
LIN {X 0,Y 331.899,Z 314.704,A -85,B 0,C 180,E1 -14668.786,E2 -14668.786} C_VEL
LIN {X 0,Y 331.903,Z 315.01,A -85,B 0,C 180,E1 -14670,E2 -14670} C_VEL
LIN {X 0,Y 331.899,Z 314.733,A -85,B 0,C 180,E1 -14671.213,E2 -14671.213} C_VEL
LIN {X 0,Y 331.964,Z 313.987,A -85,B 0,C 180,E1 -14672.426,E2 -14672.426} C_VEL
LIN {X 0,Y 332.113,Z 312.772,A -85,B 0,C 180,E1 -14673.64,E2 -14673.64} C_VEL
LIN {X 0,Y 332.414,Z 309.919,A -85,B 0,C 180,E1 -14675.459,E2 -14675.459} C_VEL
LIN {X 0,Y 332.609,Z 307.181,A -85,B 0,C 180,E1 -14676.731,E2 -14676.731} C_VEL
LIN {X 0,Y 333.114,Z 302.215,A -85,B 0,C 180,E1 -14678.492,E2 -14678.492} C_VEL
LIN {X 0,Y 333.681,Z 296.717,A -85,B 0,C 180,E1 -14680.006,E2 -14680.006} C_VEL
LIN {X 0,Y 334.499,Z 289.808,A -85,B 0,C 180,E1 -14681.513,E2 -14681.513} C_VEL
LIN {X 0,Y 335.377,Z 281.873,A -85,B 0,C 180,E1 -14682.865,E2 -14682.865} C_VEL
LIN {X 0,Y 336.161,Z 274.307,A -85,B 0,C 180,E1 -14683.911,E2 -14683.911} C_VEL
LIN {X 0,Y 336.949,Z 266.374,A -85,B 0,C 180,E1 -14684.803,E2 -14684.803} C_VEL
LIN {X 0,Y 337.377,Z 260.054,A -85,B 0,C 180,E1 -14685.402,E2 -14685.402} C_VEL
LIN {X 0,Y 338.081,Z 251.087,A -85,B 0,C 180,E1 -14686.065,E2 -14686.065} C_VEL
LIN {X 0,Y 338.517,Z 241.734,A -85,B 0,C 180,E1 -14686.586,E2 -14686.586} C_VEL
LIN {X 0,Y 338.856,Z 232.667,A -85,B 0,C 180,E1 -14686.932,E2 -14686.932} C_VEL
LIN {X 0,Y 339.293,Z 199.553,A -85,B 0,C 180,E1 -14687.668,E2 -14687.668} C_VEL
LIN {X 0,Y 339.571,Z 180.614,A -85,B 0,C 180,E1 -14688.066,E2 -14688.066} C_VEL
LIN {X 0,Y 335.114,Z 156.514,A -85,B 0,C 180,E1 -14688.859,E2 -14688.859} C_VEL
LIN {X 0,Y 335.079,Z 155.288,A -85,B 0,C 180,E1 -14689.051,E2 -14689.051} C_VEL
LIN {X 0,Y 335.07,Z 149.643,A -85,B 0,C 180,E1 -14690.889,E2 -14690.889} C_VEL
LIN {X 0,Y 333.75,Z 141.832,A -85,B 0,C 180,E1 -14693.645,E2 -14693.645} C_VEL
LIN {X 0,Y 333.744,Z 141.722,A -85,B 0,C 180,E1 -14697.598,E2 -14697.598} C_VEL
LIN {X 0,Y 333.697,Z 141.731,A -85,B 0,C 180,E1 -14700.362,E2 -14700.362} C_VEL
LIN {X 0,Y 333.641,Z 141.736,A -85,B 0,C 180,E1 -14702.71,E2 -14702.71} C_VEL
LIN {X 0,Y 332.959,Z 141.822,A -85,B 0,C 180,E1 -14703.717,E2 -14703.717} C_VEL
LIN {X 0,Y 330.103,Z 142.17,A -85,B 0,C 180,E1 -14705.355,E2 -14705.355} C_VEL
LIN {X 0,Y 327.7,Z 142.475,A -85,B 0,C 180,E1 -14706.682,E2 -14706.682} C_VEL
LIN {X 0,Y 326.68,Z 142.604,A -85,B 0,C 180,E1 -14707.709,E2 -14707.709} C_VEL
LIN {X 0,Y 326.603,Z 142.609,A -85,B 0,C 180,E1 -14708.057,E2 -14708.057} C_VEL
LIN {X 0,Y 326.575,Z 142.61,A -85,B 0,C 180,E1 -14711.845,E2 -14711.845} C_VEL
LIN {X 0,Y 326.527,Z 142.62,A -85,B 0,C 180,E1 -14715.257,E2 -14715.257} C_VEL
LIN {X 0,Y 326.576,Z 142.615,A -85,B 0,C 180,E1 -14718.868,E2 -14718.868} C_VEL
LIN {X 0,Y 326.626,Z 142.61,A -85,B 0,C 180,E1 -14722.761,E2 -14722.761} C_VEL
LIN {X 0,Y 326.606,Z 142.608,A -85,B 0,C 180,E1 -14725.98,E2 -14725.98} C_VEL
LIN {X 0,Y 326.659,Z 142.605,A -85,B 0,C 180,E1 -14730.341,E2 -14730.341} C_VEL
LIN {X 0,Y 326.689,Z 142.599,A -85,B 0,C 180,E1 -14734.516,E2 -14734.516} C_VEL
LIN {X 0,Y 326.647,Z 142.609,A -85,B 0,C 180,E1 -14738.545,E2 -14738.545} C_VEL
LIN {X 0,Y 326.743,Z 142.59,A -85,B 0,C 180,E1 -14741.177,E2 -14741.177} C_VEL
LIN {X 0,Y 326.762,Z 142.592,A -85,B 0,C 180,E1 -14745.433,E2 -14745.433} C_VEL
LIN {X 0,Y 326.772,Z 142.59,A -85,B 0,C 180,E1 -14748.839,E2 -14748.839} C_VEL
LIN {X 0,Y 326.978,Z 142.565,A -85,B 0,C 180,E1 -14752.59,E2 -14752.59} C_VEL
LIN {X 0,Y 326.776,Z 142.59,A -85,B 0,C 180,E1 -14755.065,E2 -14755.065} C_VEL
LIN {X 0,Y 327.046,Z 142.557,A -85,B 0,C 180,E1 -14757.537,E2 -14757.537} C_VEL
LIN {X 0,Y 327.197,Z 142.537,A -85,B 0,C 180,E1 -14760,E2 -14760} C_VEL
LIN {X 0,Y 327.045,Z 142.555,A -85,B 0,C 180,E1 -14762.463,E2 -14762.463} C_VEL
LIN {X 0,Y 326.997,Z 142.564,A -85,B 0,C 180,E1 -14766.169,E2 -14766.169} C_VEL
LIN {X 0,Y 326.913,Z 142.571,A -85,B 0,C 180,E1 -14768.655,E2 -14768.655} C_VEL
LIN {X 0,Y 326.733,Z 142.594,A -85,B 0,C 180,E1 -14772.421,E2 -14772.421} C_VEL
LIN {X 0,Y 326.752,Z 142.595,A -85,B 0,C 180,E1 -14774.957,E2 -14774.957} C_VEL
LIN {X 0,Y 326.731,Z 142.595,A -85,B 0,C 180,E1 -14778.838,E2 -14778.838} C_VEL
LIN {X 0,Y 326.619,Z 142.612,A -85,B 0,C 180,E1 -14782.787,E2 -14782.787} C_VEL
LIN {X 0,Y 326.688,Z 142.601,A -85,B 0,C 180,E1 -14785.484,E2 -14785.484} C_VEL
LIN {X 0,Y 326.658,Z 142.604,A -85,B 0,C 180,E1 -14789.659,E2 -14789.659} C_VEL
LIN {X 0,Y 326.605,Z 142.61,A -85,B 0,C 180,E1 -14794.02,E2 -14794.02} C_VEL
LIN {X 0,Y 326.625,Z 142.61,A -85,B 0,C 180,E1 -14797.239,E2 -14797.239} C_VEL
LIN {X 0,Y 326.575,Z 142.611,A -85,B 0,C 180,E1 -14801.131,E2 -14801.131} C_VEL
LIN {X 0,Y 326.525,Z 142.619,A -85,B 0,C 180,E1 -14804.743,E2 -14804.743} C_VEL
LIN {X 0,Y 326.574,Z 142.62,A -85,B 0,C 180,E1 -14808.154,E2 -14808.154} C_VEL
LIN {X 0,Y 326.596,Z 142.609,A -85,B 0,C 180,E1 -14811.388,E2 -14811.388} C_VEL
LIN {X 0,Y 326.618,Z 142.611,A -85,B 0,C 180,E1 -14814.852,E2 -14814.852} C_VEL
LIN {X 0,Y 326.608,Z 142.61,A -85,B 0,C 180,E1 -14817.456,E2 -14817.456} C_VEL
LIN {X 0,Y 326.659,Z 142.601,A -85,B 0,C 180,E1 -14820.341,E2 -14820.341} C_VEL
LIN {X 0,Y 326.762,Z 142.69,A -85,B 0,C 180,E1 -14822.89,E2 -14822.89} C_VEL
LIN {X 0,Y 328.418,Z 151.781,A -85,B 0,C 180,E1 -14826.01,E2 -14826.01} C_VEL
LIN {X 0,Y 328.937,Z 155.985,A -85,B 0,C 180,E1 -14827.382,E2 -14827.382} C_VEL
LIN {X 0,Y 327.864,Z 166.842,A -85,B 0,C 180,E1 -14830.669,E2 -14830.669} C_VEL
LIN {X 0,Y 328.384,Z 170.536,A -85,B 0,C 180,E1 -14830.855,E2 -14830.855} C_VEL
LIN {X 0,Y 331.949,Z 192.951,A -85,B 0,C 180,E1 -14831.568,E2 -14831.568} C_VEL
LIN {X 0,Y 332.622,Z 199.764,A -85,B 0,C 180,E1 -14831.758,E2 -14831.758} C_VEL
LIN {X 0,Y 331.953,Z 243.229,A -85,B 0,C 180,E1 -14832.719,E2 -14832.719} C_VEL
LIN {X 0,Y 331.524,Z 252.386,A -85,B 0,C 180,E1 -14833.053,E2 -14833.053} C_VEL
LIN {X 0,Y 330.942,Z 262.012,A -85,B 0,C 180,E1 -14833.578,E2 -14833.578} C_VEL
LIN {X 0,Y 330.221,Z 271.15,A -85,B 0,C 180,E1 -14834.255,E2 -14834.255} C_VEL
LIN {X 0,Y 329.285,Z 281.93,A -85,B 0,C 180,E1 -14835.319,E2 -14835.319} C_VEL
LIN {X 0,Y 328.33,Z 290.205,A -85,B 0,C 180,E1 -14836.382,E2 -14836.382} C_VEL
LIN {X 0,Y 327.474,Z 297.892,A -85,B 0,C 180,E1 -14837.608,E2 -14837.608} C_VEL
LIN {X 0,Y 326.761,Z 304.219,A -85,B 0,C 180,E1 -14838.839,E2 -14838.839} C_VEL
LIN {X 0,Y 326.183,Z 309.477,A -85,B 0,C 180,E1 -14840.075,E2 -14840.075} C_VEL
LIN {X 0,Y 325.718,Z 313.861,A -85,B 0,C 180,E1 -14841.313,E2 -14841.313} C_VEL
LIN {X 0,Y 325.264,Z 319.033,A -85,B 0,C 180,E1 -14843.175,E2 -14843.175} C_VEL
LIN {X 0,Y 324.973,Z 322.83,A -85,B 0,C 180,E1 -14845.038,E2 -14845.038} C_VEL
LIN {X 0,Y 324.92,Z 324.576,A -85,B 0,C 180,E1 -14846.28,E2 -14846.28} C_VEL
LIN {X 0,Y 324.822,Z 325.824,A -85,B 0,C 180,E1 -14847.52,E2 -14847.52} C_VEL
LIN {X 0,Y 324.781,Z 326.6,A -85,B 0,C 180,E1 -14848.76,E2 -14848.76} C_VEL
LIN {X 0,Y 324.806,Z 326.893,A -85,B 0,C 180,E1 -14850,E2 -14850} C_VEL
LIN {X 0,Y 324.781,Z 326.594,A -85,B 0,C 180,E1 -14851.24,E2 -14851.24} C_VEL
LIN {X 0,Y 324.823,Z 325.808,A -85,B 0,C 180,E1 -14852.48,E2 -14852.48} C_VEL
LIN {X 0,Y 324.92,Z 324.549,A -85,B 0,C 180,E1 -14853.721,E2 -14853.721} C_VEL
LIN {X 0,Y 324.992,Z 321.858,A -85,B 0,C 180,E1 -14855.465,E2 -14855.465} C_VEL
LIN {X 0,Y 325.264,Z 318.984,A -85,B 0,C 180,E1 -14856.825,E2 -14856.825} C_VEL
LIN {X 0,Y 325.659,Z 313.795,A -85,B 0,C 180,E1 -14858.689,E2 -14858.689} C_VEL
LIN {X 0,Y 326.451,Z 306.959,A -85,B 0,C 180,E1 -14860.544,E2 -14860.544} C_VEL
LIN {X 0,Y 327.294,Z 299.489,A -85,B 0,C 180,E1 -14862.085,E2 -14862.085} C_VEL
LIN {X 0,Y 328.136,Z 292.121,A -85,B 0,C 180,E1 -14863.312,E2 -14863.312} C_VEL
LIN {X 0,Y 328.983,Z 284.231,A -85,B 0,C 180,E1 -14864.38,E2 -14864.38} C_VEL
LIN {X 0,Y 329.785,Z 275.891,A -85,B 0,C 180,E1 -14865.291,E2 -14865.291} C_VEL
LIN {X 0,Y 330.685,Z 265.23,A -85,B 0,C 180,E1 -14866.197,E2 -14866.197} C_VEL
LIN {X 0,Y 331.416,Z 253.604,A -85,B 0,C 180,E1 -14866.874,E2 -14866.874} C_VEL
LIN {X 0,Y 331.931,Z 243.837,A -85,B 0,C 180,E1 -14867.243,E2 -14867.243} C_VEL
LIN {X 0,Y 332.416,Z 196.616,A -85,B 0,C 180,E1 -14868.302,E2 -14868.302} C_VEL
LIN {X 0,Y 328.638,Z 171.824,A -85,B 0,C 180,E1 -14869.079,E2 -14869.079} C_VEL
LIN {X 0,Y 327.846,Z 167.108,A -85,B 0,C 180,E1 -14869.274,E2 -14869.274} C_VEL
LIN {X 0,Y 328.204,Z 163.229,A -85,B 0,C 180,E1 -14870.363,E2 -14870.363} C_VEL
LIN {X 0,Y 328.911,Z 155.91,A -85,B 0,C 180,E1 -14872.62,E2 -14872.62} C_VEL
LIN {X 0,Y 328.051,Z 149.597,A -85,B 0,C 180,E1 -14874.693,E2 -14874.693} C_VEL
LIN {X 0,Y 326.744,Z 142.636,A -85,B 0,C 180,E1 -14877.134,E2 -14877.134} C_VEL
LIN {X 0,Y 326.594,Z 142.614,A -85,B 0,C 180,E1 -14881.095,E2 -14881.095} C_VEL
LIN {X 0,Y 326.607,Z 142.611,A -85,B 0,C 180,E1 -14884.02,E2 -14884.02} C_VEL
LIN {X 0,Y 326.628,Z 142.607,A -85,B 0,C 180,E1 -14887.239,E2 -14887.239} C_VEL
LIN {X 0,Y 326.578,Z 142.615,A -85,B 0,C 180,E1 -14891.132,E2 -14891.132} C_VEL
LIN {X 0,Y 326.527,Z 142.617,A -85,B 0,C 180,E1 -14894.743,E2 -14894.743} C_VEL
LIN {X 0,Y 326.576,Z 142.612,A -85,B 0,C 180,E1 -14898.154,E2 -14898.154} C_VEL
LIN {X 0,Y 326.624,Z 142.613,A -85,B 0,C 180,E1 -14901.392,E2 -14901.392} C_VEL
LIN {X 0,Y 326.62,Z 142.609,A -85,B 0,C 180,E1 -14904.852,E2 -14904.852} C_VEL
LIN {X 0,Y 326.608,Z 142.615,A -85,B 0,C 180,E1 -14907.456,E2 -14907.456} C_VEL
LIN {X 0,Y 326.661,Z 142.604,A -85,B 0,C 180,E1 -14910.341,E2 -14910.341} C_VEL
LIN {X 0,Y 326.691,Z 142.601,A -85,B 0,C 180,E1 -14914.517,E2 -14914.517} C_VEL
LIN {X 0,Y 326.65,Z 142.607,A -85,B 0,C 180,E1 -14918.546,E2 -14918.546} C_VEL
LIN {X 0,Y 326.746,Z 142.593,A -85,B 0,C 180,E1 -14921.178,E2 -14921.178} C_VEL
LIN {X 0,Y 326.765,Z 142.592,A -85,B 0,C 180,E1 -14925.433,E2 -14925.433} C_VEL
LIN {X 0,Y 326.771,Z 142.587,A -85,B 0,C 180,E1 -14928.839,E2 -14928.839} C_VEL
LIN {X 0,Y 326.96,Z 142.57,A -85,B 0,C 180,E1 -14932.59,E2 -14932.59} C_VEL
LIN {X 0,Y 326.776,Z 142.59,A -85,B 0,C 180,E1 -14935.065,E2 -14935.065} C_VEL
LIN {X 0,Y 327.047,Z 142.555,A -85,B 0,C 180,E1 -14937.537,E2 -14937.537} C_VEL
LIN {X 0,Y 327.181,Z 142.538,A -85,B 0,C 180,E1 -14940,E2 -14940} C_VEL
LIN {X 0,Y 327.047,Z 142.557,A -85,B 0,C 180,E1 -14942.463,E2 -14942.463} C_VEL
LIN {X 0,Y 326.973,Z 142.564,A -85,B 0,C 180,E1 -14946.648,E2 -14946.648} C_VEL
LIN {X 0,Y 326.818,Z 142.586,A -85,B 0,C 180,E1 -14949.906,E2 -14949.906} C_VEL
LIN {X 0,Y 326.762,Z 142.596,A -85,B 0,C 180,E1 -14953.685,E2 -14953.685} C_VEL
LIN {X 0,Y 326.701,Z 142.598,A -85,B 0,C 180,E1 -14957.528,E2 -14957.528} C_VEL
LIN {X 0,Y 326.667,Z 142.602,A -85,B 0,C 180,E1 -14960.135,E2 -14960.135} C_VEL
LIN {X 0,Y 326.654,Z 142.604,A -85,B 0,C 180,E1 -14964.129,E2 -14964.129} C_VEL
LIN {X 0,Y 326.686,Z 142.601,A -85,B 0,C 180,E1 -14966.858,E2 -14966.858} C_VEL
LIN {X 0,Y 326.641,Z 142.61,A -85,B 0,C 180,E1 -14970.611,E2 -14970.611} C_VEL
LIN {X 0,Y 326.609,Z 142.607,A -85,B 0,C 180,E1 -14974.019,E2 -14974.019} C_VEL
LIN {X 0,Y 326.629,Z 142.61,A -85,B 0,C 180,E1 -14977.239,E2 -14977.239} C_VEL
LIN {X 0,Y 326.579,Z 142.615,A -85,B 0,C 180,E1 -14981.131,E2 -14981.131} C_VEL
LIN {X 0,Y 326.529,Z 142.621,A -85,B 0,C 180,E1 -14984.743,E2 -14984.743} C_VEL
LIN {X 0,Y 326.578,Z 142.61,A -85,B 0,C 180,E1 -14988.154,E2 -14988.154} C_VEL
LIN {X 0,Y 326.626,Z 142.609,A -85,B 0,C 180,E1 -14991.391,E2 -14991.391} C_VEL
LIN {X 0,Y 326.621,Z 142.603,A -85,B 0,C 180,E1 -14994.851,E2 -14994.851} C_VEL
LIN {X 0,Y 326.612,Z 142.612,A -85,B 0,C 180,E1 -14997.456,E2 -14997.456} C_VEL
LIN {X 0,Y 326.662,Z 142.606,A -85,B 0,C 180,E1 -15000.341,E2 -15000.341} C_VEL
LIN {X 0,Y 326.692,Z 142.603,A -85,B 0,C 180,E1 -15004.516,E2 -15004.516} C_VEL
LIN {X 0,Y 326.687,Z 142.794,A -85,B 0,C 180,E1 -15006.253,E2 -15006.253} C_VEL
LIN {X 0,Y 327.943,Z 149.425,A -85,B 0,C 180,E1 -15008.634,E2 -15008.634} C_VEL
LIN {X 0,Y 328.133,Z 155.308,A -85,B 0,C 180,E1 -15010.61,E2 -15010.61} C_VEL
LIN {X 0,Y 328.225,Z 156.645,A -85,B 0,C 180,E1 -15010.838,E2 -15010.838} C_VEL
LIN {X 0,Y 332.552,Z 179.807,A -85,B 0,C 180,E1 -15011.63,E2 -15011.63} C_VEL
LIN {X 0,Y 332.803,Z 184.365,A -85,B 0,C 180,E1 -15011.746,E2 -15011.746} C_VEL
LIN {X 0,Y 331.991,Z 232.189,A -85,B 0,C 180,E1 -15012.8,E2 -15012.8} C_VEL
LIN {X 0,Y 331.626,Z 242.01,A -85,B 0,C 180,E1 -15013.177,E2 -15013.177} C_VEL
LIN {X 0,Y 331.093,Z 253.116,A -85,B 0,C 180,E1 -15013.823,E2 -15013.823} C_VEL
LIN {X 0,Y 330.221,Z 263.945,A -85,B 0,C 180,E1 -15014.729,E2 -15014.729} C_VEL
LIN {X 0,Y 329.404,Z 272.342,A -85,B 0,C 180,E1 -15015.639,E2 -15015.639} C_VEL
LIN {X 0,Y 328.676,Z 280.265,A -85,B 0,C 180,E1 -15016.711,E2 -15016.711} C_VEL
LIN {X 0,Y 327.989,Z 285.958,A -85,B 0,C 180,E1 -15017.627,E2 -15017.627} C_VEL
LIN {X 0,Y 327.275,Z 292.311,A -85,B 0,C 180,E1 -15018.856,E2 -15018.856} C_VEL
LIN {X 0,Y 326.437,Z 298.763,A -85,B 0,C 180,E1 -15020.395,E2 -15020.395} C_VEL
LIN {X 0,Y 325.947,Z 303.907,A -85,B 0,C 180,E1 -15021.943,E2 -15021.943} C_VEL
LIN {X 0,Y 325.443,Z 308.668,A -85,B 0,C 180,E1 -15023.801,E2 -15023.801} C_VEL
LIN {X 0,Y 325.254,Z 310.989,A -85,B 0,C 180,E1 -15025.041,E2 -15025.041} C_VEL
LIN {X 0,Y 325.051,Z 312.756,A -85,B 0,C 180,E1 -15026.281,E2 -15026.281} C_VEL
LIN {X 0,Y 324.886,Z 314.029,A -85,B 0,C 180,E1 -15027.52,E2 -15027.52} C_VEL
LIN {X 0,Y 324.811,Z 314.833,A -85,B 0,C 180,E1 -15028.76,E2 -15028.76} C_VEL
LIN {X 0,Y 324.811,Z 315.139,A -85,B 0,C 180,E1 -15030,E2 -15030} C_VEL
LIN {X 0,Y 324.81,Z 314.862,A -85,B 0,C 180,E1 -15031.24,E2 -15031.24} C_VEL
LIN {X 0,Y 324.885,Z 314.115,A -85,B 0,C 180,E1 -15032.479,E2 -15032.479} C_VEL
LIN {X 0,Y 325.047,Z 312.9,A -85,B 0,C 180,E1 -15033.719,E2 -15033.719} C_VEL
LIN {X 0,Y 325.35,Z 310.047,A -85,B 0,C 180,E1 -15035.578,E2 -15035.578} C_VEL
LIN {X 0,Y 325.508,Z 307.756,A -85,B 0,C 180,E1 -15036.694,E2 -15036.694} C_VEL
LIN {X 0,Y 325.936,Z 304.246,A -85,B 0,C 180,E1 -15038.057,E2 -15038.057} C_VEL
LIN {X 0,Y 326.418,Z 299.182,A -85,B 0,C 180,E1 -15039.605,E2 -15039.605} C_VEL
LIN {X 0,Y 327.044,Z 294.23,A -85,B 0,C 180,E1 -15040.838,E2 -15040.838} C_VEL
LIN {X 0,Y 327.73,Z 288.254,A -85,B 0,C 180,E1 -15042.068,E2 -15042.068} C_VEL
LIN {X 0,Y 328.553,Z 280.98,A -85,B 0,C 180,E1 -15043.294,E2 -15043.294} C_VEL
LIN {X 0,Y 329.375,Z 273.204,A -85,B 0,C 180,E1 -15044.362,E2 -15044.362} C_VEL
LIN {X 0,Y 330.202,Z 264.999,A -85,B 0,C 180,E1 -15045.271,E2 -15045.271} C_VEL
LIN {X 0,Y 330.899,Z 256.433,A -85,B 0,C 180,E1 -15046.028,E2 -15046.028} C_VEL
LIN {X 0,Y 331.619,Z 245.083,A -85,B 0,C 180,E1 -15046.783,E2 -15046.783} C_VEL
LIN {X 0,Y 332.043,Z 233.702,A -85,B 0,C 180,E1 -15047.262,E2 -15047.262} C_VEL
LIN {X 0,Y 332.377,Z 210.608,A -85,B 0,C 180,E1 -15047.805,E2 -15047.805} C_VEL
LIN {X 0,Y 332.822,Z 181.419,A -85,B 0,C 180,E1 -15048.429,E2 -15048.429} C_VEL
LIN {X 0,Y 328.193,Z 156.467,A -85,B 0,C 180,E1 -15049.286,E2 -15049.286} C_VEL
LIN {X 0,Y 328.151,Z 155.154,A -85,B 0,C 180,E1 -15049.55,E2 -15049.55} C_VEL
LIN {X 0,Y 327.986,Z 149.765,A -85,B 0,C 180,E1 -15051.362,E2 -15051.362} C_VEL
LIN {X 0,Y 326.682,Z 142.698,A -85,B 0,C 180,E1 -15053.957,E2 -15053.957} C_VEL
LIN {X 0,Y 326.685,Z 142.602,A -85,B 0,C 180,E1 -15056.857,E2 -15056.857} C_VEL
LIN {X 0,Y 326.639,Z 142.609,A -85,B 0,C 180,E1 -15060.611,E2 -15060.611} C_VEL
LIN {X 0,Y 326.608,Z 142.611,A -85,B 0,C 180,E1 -15064.019,E2 -15064.019} C_VEL
LIN {X 0,Y 326.603,Z 142.609,A -85,B 0,C 180,E1 -15068.057,E2 -15068.057} C_VEL
LIN {X 0,Y 325.958,Z 142.693,A -85,B 0,C 180,E1 -15069.087,E2 -15069.087} C_VEL
LIN {X 0,Y 323.134,Z 143.043,A -85,B 0,C 180,E1 -15070.762,E2 -15070.762} C_VEL
LIN {X 0,Y 320.703,Z 143.341,A -85,B 0,C 180,E1 -15072.12,E2 -15072.12} C_VEL
LIN {X 0,Y 319.623,Z 143.473,A -85,B 0,C 180,E1 -15073.17,E2 -15073.17} C_VEL
LIN {X 0,Y 319.515,Z 143.485,A -85,B 0,C 180,E1 -15073.527,E2 -15073.527} C_VEL
LIN {X 0,Y 319.553,Z 143.491,A -85,B 0,C 180,E1 -15077.016,E2 -15077.016} C_VEL
LIN {X 0,Y 319.546,Z 143.488,A -85,B 0,C 180,E1 -15080.371,E2 -15080.371} C_VEL
LIN {X 0,Y 319.557,Z 143.493,A -85,B 0,C 180,E1 -15083.572,E2 -15083.572} C_VEL
LIN {X 0,Y 319.576,Z 143.484,A -85,B 0,C 180,E1 -15086.686,E2 -15086.686} C_VEL
LIN {X 0,Y 319.59,Z 143.487,A -85,B 0,C 180,E1 -15089.616,E2 -15089.616} C_VEL
LIN {X 0,Y 319.607,Z 143.482,A -85,B 0,C 180,E1 -15092.498,E2 -15092.498} C_VEL
LIN {X 0,Y 319.604,Z 143.485,A -85,B 0,C 180,E1 -15095.304,E2 -15095.304} C_VEL
